// TIA Portal V20 export
// export: Created 2025-12-01T14:57:42.6383324Z, ExportSetting None, DisplayName Totally Integrated Automation Portal, DisplayVersion V20 Update 3, DisplayName TIA Portal Openness, DisplayVersion V20 Update 3, DisplayName TIA Portal Version Control Interface, DisplayVersion V20 Update 3, DisplayName STEP 7 Professional, DisplayVersion V20 Update 3, DisplayName STEP 7 Safety, DisplayVersion V20 Update 2, DisplayName WinCC Basic/Comfort/Advanced, DisplayVersion V20 Update 3, DisplayName WinCC Professional, DisplayVersion V20 Update 3, DisplayName WinCC Unified, DisplayVersion V20 Update 3
DATA_BLOCK "DB6_Recepcion"   // DB6
{ S7_Optimized_Access := 'FALSE' }
// stored: AutoNumber false
   VAR
      ByteLIbre_000 : Byte;
      FinLote_M1 : Bool;
      Especial_M1 : Bool;
      Bit_02_M1 : Bool;
      Retroceder_M1 : Bool;
      Retirar_M1 : Bool;
      Continuar_M1 : Bool;
      Entrar_M1 : Bool;
      EmiOK_M1 : Bool;
      FinLote_M2 : Bool;
      Especial_M2 : Bool;
      Bit_02_M2 : Bool;
      Retroceder_M2 : Bool;
      Retirar_M2 : Bool;
      Continuar_M2 : Bool;
      Entrar_M2 : Bool;
      EmiOK_M2 : Bool;
      FinLote_M3 : Bool;
      Especial_M3 : Bool;
      Bit_02_M3 : Bool;
      Retroceder_M3 : Bool;
      Retirar_M3 : Bool;
      Continuar_M3 : Bool;
      Entrar_M3 : Bool;
      EmiOK_M3 : Bool;
      FinLote_M4 : Bool;
      Especial_M4 : Bool;
      Bit_02_M4 : Bool;
      Retroceder_M4 : Bool;
      Retirar_M4 : Bool;
      Continuar_M4 : Bool;
      Entrar_M4 : Bool;
      EmiOK_M4 : Bool;
      FinLote_M5 : Bool;
      Especial_M5 : Bool;
      Bit_02_M5 : Bool;
      Retroceder_M5 : Bool;
      Retirar_M5 : Bool;
      Continuar_M5 : Bool;
      Entrar_M5 : Bool;
      EmiOK_M5 : Bool;
      FinLote_M6 : Bool;
      Especial_M6 : Bool;
      Bit_02_M6 : Bool;
      Retroceder_M6 : Bool;
      Retirar_M6 : Bool;
      Continuar_M6 : Bool;
      Entrar_M6 : Bool;
      EmiOK_M6 : Bool;
      FinLote_M7 : Bool;
      Especial_M7 : Bool;
      Bit_02_M7 : Bool;
      Retroceder_M7 : Bool;
      Retirar_M7 : Bool;
      Continuar_M7 : Bool;
      Entrar_M7 : Bool;
      EmiOK_M7 : Bool;
      FinLote_M8 : Bool;
      Especial_M8 : Bool;
      Bit_02_M8 : Bool;
      Retroceder_M8 : Bool;
      Retirar_M8 : Bool;
      Continuar_M8 : Bool;
      Entrar_M8 : Bool;
      EmiOK_M8 : Bool;
      FinLote_M9 : Bool;
      Especial_M9 : Bool;
      Bit_02_M9 : Bool;
      Retroceder_M9 : Bool;
      Retirar_M9 : Bool;
      Continuar_M9 : Bool;
      Entrar_M9 : Bool;
      EmiOK_M9 : Bool;
      FinLote_M10 : Bool;
      Especial_M10 : Bool;
      Bit_02_M10 : Bool;
      Retroceder_M10 : Bool;
      Retirar_M10 : Bool;
      Continuar_M10 : Bool;
      Entrar_M10 : Bool;
      EmiOK_M10 : Bool;
      FinLote_M11 : Bool;
      Especial_M11 : Bool;
      Bit_02_M11 : Bool;
      Retroceder_M11 : Bool;
      Retirar_M11 : Bool;
      Continuar_M11 : Bool;
      Entrar_M11 : Bool;
      EmiOK_M11 : Bool;
      FinLote_M12 : Bool;
      Especial_M12 : Bool;
      Bit_02_M12 : Bool;
      Retroceder_M12 : Bool;
      Retirar_M12 : Bool;
      Continuar_M12 : Bool;
      Entrar_M12 : Bool;
      EmiOK_M12 : Bool;
      FinLote_M13 : Bool;
      Especial_M13 : Bool;
      Bit_02_M13 : Bool;
      Retroceder_M13 : Bool;
      Retirar_M13 : Bool;
      Continuar_M13 : Bool;
      Entrar_M13 : Bool;
      EmiOK_M13 : Bool;
      FinLote_M14 : Bool;
      Especial_M14 : Bool;
      Bit_02_M14 : Bool;
      Retroceder_M14 : Bool;
      Retirar_M14 : Bool;
      Continuar_M14 : Bool;
      Entrar_M14 : Bool;
      EmiOK_M14 : Bool;
      FinLote_M15 : Bool;
      Especial_M15 : Bool;
      Bit_02_M15 : Bool;
      Retroceder_M15 : Bool;
      Retirar_M15 : Bool;
      Continuar_M15 : Bool;
      Entrar_M15 : Bool;
      EmiOK_M15 : Bool;
      FinLote_M16 : Bool;
      Especial_M16 : Bool;
      Bit_02_M16 : Bool;
      Retroceder_M16 : Bool;
      Retirar_M16 : Bool;
      Continuar_M16 : Bool;
      Entrar_M16 : Bool;
      EmiOK_M16 : Bool;
      FinLote_M17 : Bool;
      Especial_M17 : Bool;
      Bit_02_M17 : Bool;
      Retroceder_M17 : Bool;
      Retirar_M17 : Bool;
      Continuar_M17 : Bool;
      Entrar_M17 : Bool;
      EmiOK_M17 : Bool;
      FinLote_M18 : Bool;
      Especial_M18 : Bool;
      Bit_02_M18 : Bool;
      Retroceder_M18 : Bool;
      Retirar_M18 : Bool;
      Continuar_M18 : Bool;
      Entrar_M18 : Bool;
      EmiOK_M18 : Bool;
      FinLote_M19 : Bool;
      Especial_M19 : Bool;
      Bit_02_M19 : Bool;
      Retroceder_M19 : Bool;
      Retirar_M19 : Bool;
      Continuar_M19 : Bool;
      Entrar_M19 : Bool;
      EmiOK_M19 : Bool;
      FinLote_M20 : Bool;
      Especial_M20 : Bool;
      Bit_02_M20 : Bool;
      Retroceder_M20 : Bool;
      Retirar_M20 : Bool;
      Continuar_M20 : Bool;
      Entrar_M20 : Bool;
      EmiOK_M20 : Bool;
      FinLote_M21 : Bool;
      Especial_M21 : Bool;
      Bit_02_M21 : Bool;
      Retroceder_M21 : Bool;
      Retirar_M21 : Bool;
      Continuar_M21 : Bool;
      Entrar_M21 : Bool;
      EmiOK_M21 : Bool;
      FinLote_M22 : Bool;
      Especial_M22 : Bool;
      Bit_02_M22 : Bool;
      Retroceder_M22 : Bool;
      Retirar_M22 : Bool;
      Continuar_M22 : Bool;
      Entrar_M22 : Bool;
      EmiOK_M22 : Bool;
      FinLote_M23 : Bool;
      Especial_M23 : Bool;
      Bit_02_M23 : Bool;
      Retroceder_M23 : Bool;
      Retirar_M23 : Bool;
      Continuar_M23 : Bool;
      Entrar_M23 : Bool;
      EmiOK_M23 : Bool;
      FinLote_M24 : Bool;
      Especial_M24 : Bool;
      Bit_02_M24 : Bool;
      Retroceder_M24 : Bool;
      Retirar_M24 : Bool;
      Continuar_M24 : Bool;
      Entrar_M24 : Bool;
      EmiOK_M24 : Bool;
      FinLote_M25 : Bool;
      Especial_M25 : Bool;
      Bit_02_M25 : Bool;
      Retroceder_M25 : Bool;
      Retirar_M25 : Bool;
      Continuar_M25 : Bool;
      Entrar_M25 : Bool;
      EmiOK_M25 : Bool;
      FinLote_M26 : Bool;
      Especial_M26 : Bool;
      Bit_02_M26 : Bool;
      Retroceder_M26 : Bool;
      Retirar_M26 : Bool;
      Continuar_M26 : Bool;
      Entrar_M26 : Bool;
      EmiOK_M26 : Bool;
      FinLote_M27 : Bool;
      Especial_M27 : Bool;
      Bit_02_M27 : Bool;
      Retroceder_M27 : Bool;
      Retirar_M27 : Bool;
      Continuar_M27 : Bool;
      Entrar_M27 : Bool;
      EmiOK_M27 : Bool;
      FinLote_M28 : Bool;
      Especial_M28 : Bool;
      Bit_02_M28 : Bool;
      Retroceder_M28 : Bool;
      Retirar_M28 : Bool;
      Continuar_M28 : Bool;
      Entrar_M28 : Bool;
      EmiOK_M28 : Bool;
      FinLote_M29 : Bool;
      Especial_M29 : Bool;
      Bit_02_M29 : Bool;
      Retroceder_M29 : Bool;
      Retirar_M29 : Bool;
      Continuar_M29 : Bool;
      Entrar_M29 : Bool;
      EmiOK_M29 : Bool;
      FinLote_M30 : Bool;
      Especial_M30 : Bool;
      Bit_02_M30 : Bool;
      Retroceder_M30 : Bool;
      Retirar_M30 : Bool;
      Continuar_M30 : Bool;
      Entrar_M30 : Bool;
      EmiOK_M30 : Bool;
      FinLote_M31 : Bool;
      Especial_M31 : Bool;
      Bit_02_M31 : Bool;
      Retroceder_M31 : Bool;
      Retirar_M31 : Bool;
      Continuar_M31 : Bool;
      Entrar_M31 : Bool;
      EmiOK_M31 : Bool;
      FinLote_M32 : Bool;
      Especial_M32 : Bool;
      Bit_02_M32 : Bool;
      Retroceder_M32 : Bool;
      Retirar_M32 : Bool;
      Continuar_M32 : Bool;
      Entrar_M32 : Bool;
      EmiOK_M32 : Bool;
      FinLote_M33 : Bool;
      Especial_M33 : Bool;
      Bit_02_M33 : Bool;
      Retroceder_M33 : Bool;
      Retirar_M33 : Bool;
      Continuar_M33 : Bool;
      Entrar_M33 : Bool;
      EmiOK_M33 : Bool;
      FinLote_M34 : Bool;
      Especial_M34 : Bool;
      Bit_02_M34 : Bool;
      Retroceder_M34 : Bool;
      Retirar_M34 : Bool;
      Continuar_M34 : Bool;
      Entrar_M34 : Bool;
      EmiOK_M34 : Bool;
      FinLote_M35 : Bool;
      Especial_M35 : Bool;
      Bit_02_M35 : Bool;
      Retroceder_M35 : Bool;
      Retirar_M35 : Bool;
      Continuar_M35 : Bool;
      Entrar_M35 : Bool;
      EmiOK_M35 : Bool;
      FinLote_M36 : Bool;
      Especial_M36 : Bool;
      Bit_02_M36 : Bool;
      Retroceder_M36 : Bool;
      Retirar_M36 : Bool;
      Continuar_M36 : Bool;
      Entrar_M36 : Bool;
      EmiOK_M36 : Bool;
      FinLote_M37 : Bool;
      Especial_M37 : Bool;
      Bit_02_M37 : Bool;
      Retroceder_M37 : Bool;
      Retirar_M37 : Bool;
      Continuar_M37 : Bool;
      Entrar_M37 : Bool;
      EmiOK_M37 : Bool;
      FinLote_M38 : Bool;
      Especial_M38 : Bool;
      Bit_02_M38 : Bool;
      Retroceder_M38 : Bool;
      Retirar_M38 : Bool;
      Continuar_M38 : Bool;
      Entrar_M38 : Bool;
      EmiOK_M38 : Bool;
      FinLote_M39 : Bool;
      Especial_M39 : Bool;
      Bit_02_M39 : Bool;
      Retroceder_M39 : Bool;
      Retirar_M39 : Bool;
      Continuar_M39 : Bool;
      Entrar_M39 : Bool;
      EmiOK_M39 : Bool;
      FinLote_M40 : Bool;
      Especial_M40 : Bool;
      Bit_02_M40 : Bool;
      Retroceder_M40 : Bool;
      Retirar_M40 : Bool;
      Continuar_M40 : Bool;
      Entrar_M40 : Bool;
      EmiOK_M40 : Bool;
      FinLote_M41 : Bool;
      Especial_M41 : Bool;
      Bit_02_M41 : Bool;
      Retroceder_M41 : Bool;
      Retirar_M41 : Bool;
      Continuar_M41 : Bool;
      Entrar_M41 : Bool;
      EmiOK_M41 : Bool;
      FinLote_M42 : Bool;
      Especial_M42 : Bool;
      Bit_02_M42 : Bool;
      Retroceder_M42 : Bool;
      Retirar_M42 : Bool;
      Continuar_M42 : Bool;
      Entrar_M42 : Bool;
      EmiOK_M42 : Bool;
      FinLote_M43 : Bool;
      Especial_M43 : Bool;
      Bit_02_M43 : Bool;
      Retroceder_M43 : Bool;
      Retirar_M43 : Bool;
      Continuar_M43 : Bool;
      Entrar_M43 : Bool;
      EmiOK_M43 : Bool;
      FinLote_M44 : Bool;
      Especial_M44 : Bool;
      Bit_02_M44 : Bool;
      Retroceder_M44 : Bool;
      Retirar_M44 : Bool;
      Continuar_M44 : Bool;
      Entrar_M44 : Bool;
      EmiOK_M44 : Bool;
      FinLote_M45 : Bool;
      Especial_M45 : Bool;
      Bit_02_M45 : Bool;
      Retroceder_M45 : Bool;
      Retirar_M45 : Bool;
      Continuar_M45 : Bool;
      Entrar_M45 : Bool;
      EmiOK_M45 : Bool;
      FinLote_M46 : Bool;
      Especial_M46 : Bool;
      Bit_02_M46 : Bool;
      Retroceder_M46 : Bool;
      Retirar_M46 : Bool;
      Continuar_M46 : Bool;
      Entrar_M46 : Bool;
      EmiOK_M46 : Bool;
      FinLote_M47 : Bool;
      Especial_M47 : Bool;
      Bit_02_M47 : Bool;
      Retroceder_M47 : Bool;
      Retirar_M47 : Bool;
      Continuar_M47 : Bool;
      Entrar_M47 : Bool;
      EmiOK_M47 : Bool;
      FinLote_M48 : Bool;
      Especial_M48 : Bool;
      Bit_02_M48 : Bool;
      Retroceder_M48 : Bool;
      Retirar_M48 : Bool;
      Continuar_M48 : Bool;
      Entrar_M48 : Bool;
      EmiOK_M48 : Bool;
      FinLote_M49 : Bool;
      Especial_M49 : Bool;
      Bit_02_M49 : Bool;
      Retroceder_M49 : Bool;
      Retirar_M49 : Bool;
      Continuar_M49 : Bool;
      Entrar_M49 : Bool;
      EmiOK_M49 : Bool;
      FinLote_M50 : Bool;
      Especial_M50 : Bool;
      Bit_02_M50 : Bool;
      Retroceder_M50 : Bool;
      Retirar_M50 : Bool;
      Continuar_M50 : Bool;
      Entrar_M50 : Bool;
      EmiOK_M50 : Bool;
      FinLote_M51 : Bool;
      Especial_M51 : Bool;
      Bit_02_M51 : Bool;
      Retroceder_M51 : Bool;
      Retirar_M51 : Bool;
      Continuar_M51 : Bool;
      Entrar_M51 : Bool;
      EmiOK_M51 : Bool;
      FinLote_M52 : Bool;
      Especial_M52 : Bool;
      Bit_02_M52 : Bool;
      Retroceder_M52 : Bool;
      Retirar_M52 : Bool;
      Continuar_M52 : Bool;
      Entrar_M52 : Bool;
      EmiOK_M52 : Bool;
      FinLote_M53 : Bool;
      Especial_M53 : Bool;
      Bit_02_M53 : Bool;
      Retroceder_M53 : Bool;
      Retirar_M53 : Bool;
      Continuar_M53 : Bool;
      Entrar_M53 : Bool;
      EmiOK_M53 : Bool;
      FinLote_M54 : Bool;
      Especial_M54 : Bool;
      Bit_02_M54 : Bool;
      Retroceder_M54 : Bool;
      Retirar_M54 : Bool;
      Continuar_M54 : Bool;
      Entrar_M54 : Bool;
      EmiOK_M54 : Bool;
      FinLote_M55 : Bool;
      Especial_M55 : Bool;
      Bit_02_M55 : Bool;
      Retroceder_M55 : Bool;
      Retirar_M55 : Bool;
      Continuar_M55 : Bool;
      Entrar_M55 : Bool;
      EmiOK_M55 : Bool;
      FinLote_M56 : Bool;
      Especial_M56 : Bool;
      Bit_02_M56 : Bool;
      Retroceder_M56 : Bool;
      Retirar_M56 : Bool;
      Continuar_M56 : Bool;
      Entrar_M56 : Bool;
      EmiOK_M56 : Bool;
      FinLote_M57 : Bool;
      Especial_M57 : Bool;
      Bit_02_M57 : Bool;
      Retroceder_M57 : Bool;
      Retirar_M57 : Bool;
      Continuar_M57 : Bool;
      Entrar_M57 : Bool;
      EmiOK_M57 : Bool;
      FinLote_M58 : Bool;
      Especial_M58 : Bool;
      Bit_02_M58 : Bool;
      Retroceder_M58 : Bool;
      Retirar_M58 : Bool;
      Continuar_M58 : Bool;
      Entrar_M58 : Bool;
      EmiOK_M58 : Bool;
      FinLote_M59 : Bool;
      Especial_M59 : Bool;
      Bit_02_M59 : Bool;
      Retroceder_M59 : Bool;
      Retirar_M59 : Bool;
      Continuar_M59 : Bool;
      Entrar_M59 : Bool;
      EmiOK_M59 : Bool;
      FinLote_M60 : Bool;
      Especial_M60 : Bool;
      Bit_02_M60 : Bool;
      Retroceder_M60 : Bool;
      Retirar_M60 : Bool;
      Continuar_M60 : Bool;
      Entrar_M60 : Bool;
      EmiOK_M60 : Bool;
      FinLote_M61 : Bool;
      Especial_M61 : Bool;
      Bit_02_M61 : Bool;
      Retroceder_M61 : Bool;
      Retirar_M61 : Bool;
      Continuar_M61 : Bool;
      Entrar_M61 : Bool;
      EmiOK_M61 : Bool;
      FinLote_M62 : Bool;
      Especial_M62 : Bool;
      Bit_02_M62 : Bool;
      Retroceder_M62 : Bool;
      Retirar_M62 : Bool;
      Continuar_M62 : Bool;
      Entrar_M62 : Bool;
      EmiOK_M62 : Bool;
      FinLote_M63 : Bool;
      Especial_M63 : Bool;
      Bit_02_M63 : Bool;
      Retroceder_M63 : Bool;
      Retirar_M63 : Bool;
      Continuar_M63 : Bool;
      Entrar_M63 : Bool;
      EmiOK_M63 : Bool;
      FinLote_M64 : Bool;
      Especial_M64 : Bool;
      Bit_02_M64 : Bool;
      Retroceder_M64 : Bool;
      Retirar_M64 : Bool;
      Continuar_M64 : Bool;
      Entrar_M64 : Bool;
      EmiOK_M64 : Bool;
      FinLote_M65 : Bool;
      Especial_M65 : Bool;
      Bit_02_M65 : Bool;
      Retroceder_M65 : Bool;
      Retirar_M65 : Bool;
      Continuar_M65 : Bool;
      Entrar_M65 : Bool;
      EmiOK_M65 : Bool;
      FinLote_M66 : Bool;
      Especial_M66 : Bool;
      Bit_02_M66 : Bool;
      Retroceder_M66 : Bool;
      Retirar_M66 : Bool;
      Continuar_M66 : Bool;
      Entrar_M66 : Bool;
      EmiOK_M66 : Bool;
      FinLote_M67 : Bool;
      Especial_M67 : Bool;
      Bit_02_M67 : Bool;
      Retroceder_M67 : Bool;
      Retirar_M67 : Bool;
      Continuar_M67 : Bool;
      Entrar_M67 : Bool;
      EmiOK_M67 : Bool;
      FinLote_M68 : Bool;
      Especial_M68 : Bool;
      Bit_02_M68 : Bool;
      Retroceder_M68 : Bool;
      Retirar_M68 : Bool;
      Continuar_M68 : Bool;
      Entrar_M68 : Bool;
      EmiOK_M68 : Bool;
      FinLote_M69 : Bool;
      Especial_M69 : Bool;
      Bit_02_M69 : Bool;
      Retroceder_M69 : Bool;
      Retirar_M69 : Bool;
      Continuar_M69 : Bool;
      Entrar_M69 : Bool;
      EmiOK_M69 : Bool;
      FinLote_M70 : Bool;
      Especial_M70 : Bool;
      Bit_02_M70 : Bool;
      Retroceder_M70 : Bool;
      Retirar_M70 : Bool;
      Continuar_M70 : Bool;
      Entrar_M70 : Bool;
      EmiOK_M70 : Bool;
      FinLote_M71 : Bool;
      Especial_M71 : Bool;
      Bit_02_M71 : Bool;
      Retroceder_M71 : Bool;
      Retirar_M71 : Bool;
      Continuar_M71 : Bool;
      Entrar_M71 : Bool;
      EmiOK_M71 : Bool;
      FinLote_M72 : Bool;
      Especial_M72 : Bool;
      Bit_02_M72 : Bool;
      Retroceder_M72 : Bool;
      Retirar_M72 : Bool;
      Continuar_M72 : Bool;
      Entrar_M72 : Bool;
      EmiOK_M72 : Bool;
      FinLote_M73 : Bool;
      Especial_M73 : Bool;
      Bit_02_M73 : Bool;
      Retroceder_M73 : Bool;
      Retirar_M73 : Bool;
      Continuar_M73 : Bool;
      Entrar_M73 : Bool;
      EmiOK_M73 : Bool;
      FinLote_M74 : Bool;
      Especial_M74 : Bool;
      Bit_02_M74 : Bool;
      Retroceder_M74 : Bool;
      Retirar_M74 : Bool;
      Continuar_M74 : Bool;
      Entrar_M74 : Bool;
      EmiOK_M74 : Bool;
      FinLote_M75 : Bool;
      Especial_M75 : Bool;
      Bit_02_M75 : Bool;
      Retroceder_M75 : Bool;
      Retirar_M75 : Bool;
      Continuar_M75 : Bool;
      Entrar_M75 : Bool;
      EmiOK_M75 : Bool;
      FinLote_M76 : Bool;
      Especial_M76 : Bool;
      Bit_02_M76 : Bool;
      Retroceder_M76 : Bool;
      Retirar_M76 : Bool;
      Continuar_M76 : Bool;
      Entrar_M76 : Bool;
      EmiOK_M76 : Bool;
      FinLote_M77 : Bool;
      Especial_M77 : Bool;
      Bit_02_M77 : Bool;
      Retroceder_M77 : Bool;
      Retirar_M77 : Bool;
      Continuar_M77 : Bool;
      Entrar_M77 : Bool;
      EmiOK_M77 : Bool;
      FinLote_M78 : Bool;
      Especial_M78 : Bool;
      Bit_02_M78 : Bool;
      Retroceder_M78 : Bool;
      Retirar_M78 : Bool;
      Continuar_M78 : Bool;
      Entrar_M78 : Bool;
      EmiOK_M78 : Bool;
      FinLote_M79 : Bool;
      Especial_M79 : Bool;
      Bit_02_M79 : Bool;
      Retroceder_M79 : Bool;
      Retirar_M79 : Bool;
      Continuar_M79 : Bool;
      Entrar_M79 : Bool;
      EmiOK_M79 : Bool;
      FinLote_M80 : Bool;
      Especial_M80 : Bool;
      Bit_02_M80 : Bool;
      Retroceder_M80 : Bool;
      Retirar_M80 : Bool;
      Continuar_M80 : Bool;
      Entrar_M80 : Bool;
      EmiOK_M80 : Bool;
      FinLote_M81 : Bool;
      Especial_M81 : Bool;
      Bit_02_M81 : Bool;
      Retroceder_M81 : Bool;
      Retirar_M81 : Bool;
      Continuar_M81 : Bool;
      Entrar_M81 : Bool;
      EmiOK_M81 : Bool;
      FinLote_M82 : Bool;
      Especial_M82 : Bool;
      Bit_02_M82 : Bool;
      Retroceder_M82 : Bool;
      Retirar_M82 : Bool;
      Continuar_M82 : Bool;
      Entrar_M82 : Bool;
      EmiOK_M82 : Bool;
      FinLote_M83 : Bool;
      Especial_M83 : Bool;
      Bit_02_M83 : Bool;
      Retroceder_M83 : Bool;
      Retirar_M83 : Bool;
      Continuar_M83 : Bool;
      Entrar_M83 : Bool;
      EmiOK_M83 : Bool;
      FinLote_M84 : Bool;
      Especial_M84 : Bool;
      Bit_02_M84 : Bool;
      Retroceder_M84 : Bool;
      Retirar_M84 : Bool;
      Continuar_M84 : Bool;
      Entrar_M84 : Bool;
      EmiOK_M84 : Bool;
      FinLote_M85 : Bool;
      Especial_M85 : Bool;
      Bit_02_M85 : Bool;
      Retroceder_M85 : Bool;
      Retirar_M85 : Bool;
      Continuar_M85 : Bool;
      Entrar_M85 : Bool;
      EmiOK_M85 : Bool;
      FinLote_M86 : Bool;
      Especial_M86 : Bool;
      Bit_02_M86 : Bool;
      Retroceder_M86 : Bool;
      Retirar_M86 : Bool;
      Continuar_M86 : Bool;
      Entrar_M86 : Bool;
      EmiOK_M86 : Bool;
      FinLote_M87 : Bool;
      Especial_M87 : Bool;
      Bit_02_M87 : Bool;
      Retroceder_M87 : Bool;
      Retirar_M87 : Bool;
      Continuar_M87 : Bool;
      Entrar_M87 : Bool;
      EmiOK_M87 : Bool;
      FinLote_M88 : Bool;
      Especial_M88 : Bool;
      Bit_02_M88 : Bool;
      Retroceder_M88 : Bool;
      Retirar_M88 : Bool;
      Continuar_M88 : Bool;
      Entrar_M88 : Bool;
      EmiOK_M88 : Bool;
      FinLote_M89 : Bool;
      Especial_M89 : Bool;
      Bit_02_M89 : Bool;
      Retroceder_M89 : Bool;
      Retirar_M89 : Bool;
      Continuar_M89 : Bool;
      Entrar_M89 : Bool;
      EmiOK_M89 : Bool;
      FinLote_M90 : Bool;
      Especial_M90 : Bool;
      Bit_02_M90 : Bool;
      Retroceder_M90 : Bool;
      Retirar_M90 : Bool;
      Continuar_M90 : Bool;
      Entrar_M90 : Bool;
      EmiOK_M90 : Bool;
      FinLote_M91 : Bool;
      Especial_M91 : Bool;
      Bit_02_M91 : Bool;
      Retroceder_M91 : Bool;
      Retirar_M91 : Bool;
      Continuar_M91 : Bool;
      Entrar_M91 : Bool;
      EmiOK_M91 : Bool;
      FinLote_M92 : Bool;
      Especial_M92 : Bool;
      Bit_02_M92 : Bool;
      Retroceder_M92 : Bool;
      Retirar_M92 : Bool;
      Continuar_M92 : Bool;
      Entrar_M92 : Bool;
      EmiOK_M92 : Bool;
      FinLote_M93 : Bool;
      Especial_M93 : Bool;
      Bit_02_M93 : Bool;
      Retroceder_M93 : Bool;
      Retirar_M93 : Bool;
      Continuar_M93 : Bool;
      Entrar_M93 : Bool;
      EmiOK_M93 : Bool;
      FinLote_M94 : Bool;
      Especial_M94 : Bool;
      Bit_02_M94 : Bool;
      Retroceder_M94 : Bool;
      Retirar_M94 : Bool;
      Continuar_M94 : Bool;
      Entrar_M94 : Bool;
      EmiOK_M94 : Bool;
      FinLote_M95 : Bool;
      Especial_M95 : Bool;
      Bit_02_M95 : Bool;
      Retroceder_M95 : Bool;
      Retirar_M95 : Bool;
      Continuar_M95 : Bool;
      Entrar_M95 : Bool;
      EmiOK_M95 : Bool;
      FinLote_M96 : Bool;
      Especial_M96 : Bool;
      Bit_02_M96 : Bool;
      Retroceder_M96 : Bool;
      Retirar_M96 : Bool;
      Continuar_M96 : Bool;
      Entrar_M96 : Bool;
      EmiOK_M96 : Bool;
      FinLote_M97 : Bool;
      Especial_M97 : Bool;
      Bit_02_M97 : Bool;
      Retroceder_M97 : Bool;
      Retirar_M97 : Bool;
      Continuar_M97 : Bool;
      Entrar_M97 : Bool;
      EmiOK_M97 : Bool;
      FinLote_M98 : Bool;
      Especial_M98 : Bool;
      Bit_02_M98 : Bool;
      Retroceder_M98 : Bool;
      Retirar_M98 : Bool;
      Continuar_M98 : Bool;
      Entrar_M98 : Bool;
      EmiOK_M98 : Bool;
      FinLote_M99 : Bool;
      Especial_M99 : Bool;
      Bit_02_M99 : Bool;
      Retroceder_M99 : Bool;
      Retirar_M99 : Bool;
      Continuar_M99 : Bool;
      Entrar_M99 : Bool;
      EmiOK_M99 : Bool;
      FinLote_M100 : Bool;
      Especial_M100 : Bool;
      Bit_02_M100 : Bool;
      Retroceder_M100 : Bool;
      Retirar_M100 : Bool;
      Continuar_M100 : Bool;
      Entrar_M100 : Bool;
      EmiOK_M100 : Bool;
      FinLote_M101 : Bool;
      Especial_M101 : Bool;
      Bit_02_M101 : Bool;
      Retroceder_M101 : Bool;
      Retirar_M101 : Bool;
      Continuar_M101 : Bool;
      Entrar_M101 : Bool;
      EmiOK_M101 : Bool;
      FinLote_M102 : Bool;
      Especial_M102 : Bool;
      Bit_02_M102 : Bool;
      Retroceder_M102 : Bool;
      Retirar_M102 : Bool;
      Continuar_M102 : Bool;
      Entrar_M102 : Bool;
      EmiOK_M102 : Bool;
      FinLote_M103 : Bool;
      Especial_M103 : Bool;
      Bit_02_M103 : Bool;
      Retroceder_M103 : Bool;
      Retirar_M103 : Bool;
      Continuar_M103 : Bool;
      Entrar_M103 : Bool;
      EmiOK_M103 : Bool;
      FinLote_M104 : Bool;
      Especial_M104 : Bool;
      Bit_02_M104 : Bool;
      Retroceder_M104 : Bool;
      Retirar_M104 : Bool;
      Continuar_M104 : Bool;
      Entrar_M104 : Bool;
      EmiOK_M104 : Bool;
      FinLote_M105 : Bool;
      Especial_M105 : Bool;
      Bit_02_M105 : Bool;
      Retroceder_M105 : Bool;
      Retirar_M105 : Bool;
      Continuar_M105 : Bool;
      Entrar_M105 : Bool;
      EmiOK_M105 : Bool;
      FinLote_M106 : Bool;
      Especial_M106 : Bool;
      Bit_02_M106 : Bool;
      Retroceder_M106 : Bool;
      Retirar_M106 : Bool;
      Continuar_M106 : Bool;
      Entrar_M106 : Bool;
      EmiOK_M106 : Bool;
      FinLote_M107 : Bool;
      Especial_M107 : Bool;
      Bit_02_M107 : Bool;
      Retroceder_M107 : Bool;
      Retirar_M107 : Bool;
      Continuar_M107 : Bool;
      Entrar_M107 : Bool;
      EmiOK_M107 : Bool;
      FinLote_M108 : Bool;
      Especial_M108 : Bool;
      Bit_02_M108 : Bool;
      Retroceder_M108 : Bool;
      Retirar_M108 : Bool;
      Continuar_M108 : Bool;
      Entrar_M108 : Bool;
      EmiOK_M108 : Bool;
      FinLote_M109 : Bool;
      Especial_M109 : Bool;
      Bit_02_M109 : Bool;
      Retroceder_M109 : Bool;
      Retirar_M109 : Bool;
      Continuar_M109 : Bool;
      Entrar_M109 : Bool;
      EmiOK_M109 : Bool;
      FinLote_M110 : Bool;
      Especial_M110 : Bool;
      Bit_02_M110 : Bool;
      Retroceder_M110 : Bool;
      Retirar_M110 : Bool;
      Continuar_M110 : Bool;
      Entrar_M110 : Bool;
      EmiOK_M110 : Bool;
      FinLote_M111 : Bool;
      Especial_M111 : Bool;
      Bit_02_M111 : Bool;
      Retroceder_M111 : Bool;
      Retirar_M111 : Bool;
      Continuar_M111 : Bool;
      Entrar_M111 : Bool;
      EmiOK_M111 : Bool;
      FinLote_M112 : Bool;
      Especial_M112 : Bool;
      Bit_02_M112 : Bool;
      Retroceder_M112 : Bool;
      Retirar_M112 : Bool;
      Continuar_M112 : Bool;
      Entrar_M112 : Bool;
      EmiOK_M112 : Bool;
      FinLote_M113 : Bool;
      Especial_M113 : Bool;
      Bit_02_M113 : Bool;
      Retroceder_M113 : Bool;
      Retirar_M113 : Bool;
      Continuar_M113 : Bool;
      Entrar_M113 : Bool;
      EmiOK_M113 : Bool;
      FinLote_M114 : Bool;
      Especial_M114 : Bool;
      Bit_02_M114 : Bool;
      Retroceder_M114 : Bool;
      Retirar_M114 : Bool;
      Continuar_M114 : Bool;
      Entrar_M114 : Bool;
      EmiOK_M114 : Bool;
      FinLote_M115 : Bool;
      Especial_M115 : Bool;
      Bit_02_M115 : Bool;
      Retroceder_M115 : Bool;
      Retirar_M115 : Bool;
      Continuar_M115 : Bool;
      Entrar_M115 : Bool;
      EmiOK_M115 : Bool;
      FinLote_M116 : Bool;
      Especial_M116 : Bool;
      Bit_02_M116 : Bool;
      Retroceder_M116 : Bool;
      Retirar_M116 : Bool;
      Continuar_M116 : Bool;
      Entrar_M116 : Bool;
      EmiOK_M116 : Bool;
      FinLote_M117 : Bool;
      Especial_M117 : Bool;
      Bit_02_M117 : Bool;
      Retroceder_M117 : Bool;
      Retirar_M117 : Bool;
      Continuar_M117 : Bool;
      Entrar_M117 : Bool;
      EmiOK_M117 : Bool;
      FinLote_M118 : Bool;
      Especial_M118 : Bool;
      Bit_02_M118 : Bool;
      Retroceder_M118 : Bool;
      Retirar_M118 : Bool;
      Continuar_M118 : Bool;
      Entrar_M118 : Bool;
      EmiOK_M118 : Bool;
      FinLote_M119 : Bool;
      Especial_M119 : Bool;
      Bit_02_M119 : Bool;
      Retroceder_M119 : Bool;
      Retirar_M119 : Bool;
      Continuar_M119 : Bool;
      Entrar_M119 : Bool;
      EmiOK_M119 : Bool;
      FinLote_M120 : Bool;
      Especial_M120 : Bool;
      Bit_02_M120 : Bool;
      Retroceder_M120 : Bool;
      Retirar_M120 : Bool;
      Continuar_M120 : Bool;
      Entrar_M120 : Bool;
      EmiOK_M120 : Bool;
      FinLote_M121 : Bool;
      Especial_M121 : Bool;
      Bit_02_M121 : Bool;
      Retroceder_M121 : Bool;
      Retirar_M121 : Bool;
      Continuar_M121 : Bool;
      Entrar_M121 : Bool;
      EmiOK_M121 : Bool;
      FinLote_M122 : Bool;
      Especial_M122 : Bool;
      Bit_02_M122 : Bool;
      Retroceder_M122 : Bool;
      Retirar_M122 : Bool;
      Continuar_M122 : Bool;
      Entrar_M122 : Bool;
      EmiOK_M122 : Bool;
      FinLote_M123 : Bool;
      Especial_M123 : Bool;
      Bit_02_M123 : Bool;
      Retroceder_M123 : Bool;
      Retirar_M123 : Bool;
      Continuar_M123 : Bool;
      Entrar_M123 : Bool;
      EmiOK_M123 : Bool;
      FinLote_M124 : Bool;
      Especial_M124 : Bool;
      Bit_02_M124 : Bool;
      Retroceder_M124 : Bool;
      Retirar_M124 : Bool;
      Continuar_M124 : Bool;
      Entrar_M124 : Bool;
      EmiOK_M124 : Bool;
      FinLote_M125 : Bool;
      Especial_M125 : Bool;
      Bit_02_M125 : Bool;
      Retroceder_M125 : Bool;
      Retirar_M125 : Bool;
      Continuar_M125 : Bool;
      Entrar_M125 : Bool;
      EmiOK_M125 : Bool;
      FinLote_M126 : Bool;
      Especial_M126 : Bool;
      Bit_02_M126 : Bool;
      Retroceder_M126 : Bool;
      Retirar_M126 : Bool;
      Continuar_M126 : Bool;
      Entrar_M126 : Bool;
      EmiOK_M126 : Bool;
      FinLote_M127 : Bool;
      Especial_M127 : Bool;
      Bit_02_M127 : Bool;
      Retroceder_M127 : Bool;
      Retirar_M127 : Bool;
      Continuar_M127 : Bool;
      Entrar_M127 : Bool;
      EmiOK_M127 : Bool;
      FinLote_M128 : Bool;
      Especial_M128 : Bool;
      Bit_02_M128 : Bool;
      Retroceder_M128 : Bool;
      Retirar_M128 : Bool;
      Continuar_M128 : Bool;
      Entrar_M128 : Bool;
      EmiOK_M128 : Bool;
      FinLote_M129 : Bool;
      Especial_M129 : Bool;
      Bit_02_M129 : Bool;
      Retroceder_M129 : Bool;
      Retirar_M129 : Bool;
      Continuar_M129 : Bool;
      Entrar_M129 : Bool;
      EmiOK_M129 : Bool;
      FinLote_M130 : Bool;
      Especial_M130 : Bool;
      Bit_02_M130 : Bool;
      Retroceder_M130 : Bool;
      Retirar_M130 : Bool;
      Continuar_M130 : Bool;
      Entrar_M130 : Bool;
      EmiOK_M130 : Bool;
      FinLote_M131 : Bool;
      Especial_M131 : Bool;
      Bit_02_M131 : Bool;
      Retroceder_M131 : Bool;
      Retirar_M131 : Bool;
      Continuar_M131 : Bool;
      Entrar_M131 : Bool;
      EmiOK_M131 : Bool;
      FinLote_M132 : Bool;
      Especial_M132 : Bool;
      Bit_02_M132 : Bool;
      Retroceder_M132 : Bool;
      Retirar_M132 : Bool;
      Continuar_M132 : Bool;
      Entrar_M132 : Bool;
      EmiOK_M132 : Bool;
      FinLote_M133 : Bool;
      Especial_M133 : Bool;
      Bit_02_M133 : Bool;
      Retroceder_M133 : Bool;
      Retirar_M133 : Bool;
      Continuar_M133 : Bool;
      Entrar_M133 : Bool;
      EmiOK_M133 : Bool;
      FinLote_M134 : Bool;
      Especial_M134 : Bool;
      Bit_02_M134 : Bool;
      Retroceder_M134 : Bool;
      Retirar_M134 : Bool;
      Continuar_M134 : Bool;
      Entrar_M134 : Bool;
      EmiOK_M134 : Bool;
      FinLote_M135 : Bool;
      Especial_M135 : Bool;
      Bit_02_M135 : Bool;
      Retroceder_M135 : Bool;
      Retirar_M135 : Bool;
      Continuar_M135 : Bool;
      Entrar_M135 : Bool;
      EmiOK_M135 : Bool;
      FinLote_M136 : Bool;
      Especial_M136 : Bool;
      Bit_02_M136 : Bool;
      Retroceder_M136 : Bool;
      Retirar_M136 : Bool;
      Continuar_M136 : Bool;
      Entrar_M136 : Bool;
      EmiOK_M136 : Bool;
      FinLote_M137 : Bool;
      Especial_M137 : Bool;
      Bit_02_M137 : Bool;
      Retroceder_M137 : Bool;
      Retirar_M137 : Bool;
      Continuar_M137 : Bool;
      Entrar_M137 : Bool;
      EmiOK_M137 : Bool;
      FinLote_M138 : Bool;
      Especial_M138 : Bool;
      Bit_02_M138 : Bool;
      Retroceder_M138 : Bool;
      Retirar_M138 : Bool;
      Continuar_M138 : Bool;
      Entrar_M138 : Bool;
      EmiOK_M138 : Bool;
      FinLote_M139 : Bool;
      Especial_M139 : Bool;
      Bit_02_M139 : Bool;
      Retroceder_M139 : Bool;
      Retirar_M139 : Bool;
      Continuar_M139 : Bool;
      Entrar_M139 : Bool;
      EmiOK_M139 : Bool;
      FinLote_M140 : Bool;
      Especial_M140 : Bool;
      Bit_02_M140 : Bool;
      Retroceder_M140 : Bool;
      Retirar_M140 : Bool;
      Continuar_M140 : Bool;
      Entrar_M140 : Bool;
      EmiOK_M140 : Bool;
      FinLote_M141 : Bool;
      Especial_M141 : Bool;
      Bit_02_M141 : Bool;
      Retroceder_M141 : Bool;
      Retirar_M141 : Bool;
      Continuar_M141 : Bool;
      Entrar_M141 : Bool;
      EmiOK_M141 : Bool;
      FinLote_M142 : Bool;
      Especial_M142 : Bool;
      Bit_02_M142 : Bool;
      Retroceder_M142 : Bool;
      Retirar_M142 : Bool;
      Continuar_M142 : Bool;
      Entrar_M142 : Bool;
      EmiOK_M142 : Bool;
      FinLote_M143 : Bool;
      Especial_M143 : Bool;
      Bit_02_M143 : Bool;
      Retroceder_M143 : Bool;
      Retirar_M143 : Bool;
      Continuar_M143 : Bool;
      Entrar_M143 : Bool;
      EmiOK_M143 : Bool;
      FinLote_M144 : Bool;
      Especial_M144 : Bool;
      Bit_02_M144 : Bool;
      Retroceder_M144 : Bool;
      Retirar_M144 : Bool;
      Continuar_M144 : Bool;
      Entrar_M144 : Bool;
      EmiOK_M144 : Bool;
      FinLote_M145 : Bool;
      Especial_M145 : Bool;
      Bit_02_M145 : Bool;
      Retroceder_M145 : Bool;
      Retirar_M145 : Bool;
      Continuar_M145 : Bool;
      Entrar_M145 : Bool;
      EmiOK_M145 : Bool;
      FinLote_M146 : Bool;
      Especial_M146 : Bool;
      Bit_02_M146 : Bool;
      Retroceder_M146 : Bool;
      Retirar_M146 : Bool;
      Continuar_M146 : Bool;
      Entrar_M146 : Bool;
      EmiOK_M146 : Bool;
      FinLote_M147 : Bool;
      Especial_M147 : Bool;
      Bit_02_M147 : Bool;
      Retroceder_M147 : Bool;
      Retirar_M147 : Bool;
      Continuar_M147 : Bool;
      Entrar_M147 : Bool;
      EmiOK_M147 : Bool;
      FinLote_M148 : Bool;
      Especial_M148 : Bool;
      Bit_02_M148 : Bool;
      Retroceder_M148 : Bool;
      Retirar_M148 : Bool;
      Continuar_M148 : Bool;
      Entrar_M148 : Bool;
      EmiOK_M148 : Bool;
      FinLote_M149 : Bool;
      Especial_M149 : Bool;
      Bit_02_M149 : Bool;
      Retroceder_M149 : Bool;
      Retirar_M149 : Bool;
      Continuar_M149 : Bool;
      Entrar_M149 : Bool;
      EmiOK_M149 : Bool;
      FinLote_M150 : Bool;
      Especial_M150 : Bool;
      Bit_02_M150 : Bool;
      Retroceder_M150 : Bool;
      Retirar_M150 : Bool;
      Continuar_M150 : Bool;
      Entrar_M150 : Bool;
      EmiOK_M150 : Bool;
      FinLote_M151 : Bool;
      Especial_M151 : Bool;
      Bit_02_M151 : Bool;
      Retroceder_M151 : Bool;
      Retirar_M151 : Bool;
      Continuar_M151 : Bool;
      Entrar_M151 : Bool;
      EmiOK_M151 : Bool;
      FinLote_M152 : Bool;
      Especial_M152 : Bool;
      Bit_02_M152 : Bool;
      Retroceder_M152 : Bool;
      Retirar_M152 : Bool;
      Continuar_M152 : Bool;
      Entrar_M152 : Bool;
      EmiOK_M152 : Bool;
      FinLote_M153 : Bool;
      Especial_M153 : Bool;
      Bit_02_M153 : Bool;
      Retroceder_M153 : Bool;
      Retirar_M153 : Bool;
      Continuar_M153 : Bool;
      Entrar_M153 : Bool;
      EmiOK_M153 : Bool;
      FinLote_M154 : Bool;
      Especial_M154 : Bool;
      Bit_02_M154 : Bool;
      Retroceder_M154 : Bool;
      Retirar_M154 : Bool;
      Continuar_M154 : Bool;
      Entrar_M154 : Bool;
      EmiOK_M154 : Bool;
      FinLote_M155 : Bool;
      Especial_M155 : Bool;
      Bit_02_M155 : Bool;
      Retroceder_M155 : Bool;
      Retirar_M155 : Bool;
      Continuar_M155 : Bool;
      Entrar_M155 : Bool;
      EmiOK_M155 : Bool;
      FinLote_M156 : Bool;
      Especial_M156 : Bool;
      Bit_02_M156 : Bool;
      Retroceder_M156 : Bool;
      Retirar_M156 : Bool;
      Continuar_M156 : Bool;
      Entrar_M156 : Bool;
      EmiOK_M156 : Bool;
      FinLote_M157 : Bool;
      Especial_M157 : Bool;
      Bit_02_M157 : Bool;
      Retroceder_M157 : Bool;
      Retirar_M157 : Bool;
      Continuar_M157 : Bool;
      Entrar_M157 : Bool;
      EmiOK_M157 : Bool;
      FinLote_M158 : Bool;
      Especial_M158 : Bool;
      Bit_02_M158 : Bool;
      Retroceder_M158 : Bool;
      Retirar_M158 : Bool;
      Continuar_M158 : Bool;
      Entrar_M158 : Bool;
      EmiOK_M158 : Bool;
      FinLote_M159 : Bool;
      Especial_M159 : Bool;
      Bit_02_M159 : Bool;
      Retroceder_M159 : Bool;
      Retirar_M159 : Bool;
      Continuar_M159 : Bool;
      Entrar_M159 : Bool;
      EmiOK_M159 : Bool;
      FinLote_M160 : Bool;
      Especial_M160 : Bool;
      Bit_02_M160 : Bool;
      Retroceder_M160 : Bool;
      Retirar_M160 : Bool;
      Continuar_M160 : Bool;
      Entrar_M160 : Bool;
      EmiOK_M160 : Bool;
      FinLote_M161 : Bool;
      Especial_M161 : Bool;
      Bit_02_M161 : Bool;
      Retroceder_M161 : Bool;
      Retirar_M161 : Bool;
      Continuar_M161 : Bool;
      Entrar_M161 : Bool;
      EmiOK_M161 : Bool;
      FinLote_M162 : Bool;
      Especial_M162 : Bool;
      Bit_02_M162 : Bool;
      Retroceder_M162 : Bool;
      Retirar_M162 : Bool;
      Continuar_M162 : Bool;
      Entrar_M162 : Bool;
      EmiOK_M162 : Bool;
      FinLote_M163 : Bool;
      Especial_M163 : Bool;
      Bit_02_M163 : Bool;
      Retroceder_M163 : Bool;
      Retirar_M163 : Bool;
      Continuar_M163 : Bool;
      Entrar_M163 : Bool;
      EmiOK_M163 : Bool;
      FinLote_M164 : Bool;
      Especial_M164 : Bool;
      Bit_02_M164 : Bool;
      Retroceder_M164 : Bool;
      Retirar_M164 : Bool;
      Continuar_M164 : Bool;
      Entrar_M164 : Bool;
      EmiOK_M164 : Bool;
      FinLote_M165 : Bool;
      Especial_M165 : Bool;
      Bit_02_M165 : Bool;
      Retroceder_M165 : Bool;
      Retirar_M165 : Bool;
      Continuar_M165 : Bool;
      Entrar_M165 : Bool;
      EmiOK_M165 : Bool;
      FinLote_M166 : Bool;
      Especial_M166 : Bool;
      Bit_02_M166 : Bool;
      Retroceder_M166 : Bool;
      Retirar_M166 : Bool;
      Continuar_M166 : Bool;
      Entrar_M166 : Bool;
      EmiOK_M166 : Bool;
      FinLote_M167 : Bool;
      Especial_M167 : Bool;
      Bit_02_M167 : Bool;
      Retroceder_M167 : Bool;
      Retirar_M167 : Bool;
      Continuar_M167 : Bool;
      Entrar_M167 : Bool;
      EmiOK_M167 : Bool;
      FinLote_M168 : Bool;
      Especial_M168 : Bool;
      Bit_02_M168 : Bool;
      Retroceder_M168 : Bool;
      Retirar_M168 : Bool;
      Continuar_M168 : Bool;
      Entrar_M168 : Bool;
      EmiOK_M168 : Bool;
      FinLote_M169 : Bool;
      Especial_M169 : Bool;
      Bit_02_M169 : Bool;
      Retroceder_M169 : Bool;
      Retirar_M169 : Bool;
      Continuar_M169 : Bool;
      Entrar_M169 : Bool;
      EmiOK_M169 : Bool;
      FinLote_M170 : Bool;
      Especial_M170 : Bool;
      Bit_02_M170 : Bool;
      Retroceder_M170 : Bool;
      Retirar_M170 : Bool;
      Continuar_M170 : Bool;
      Entrar_M170 : Bool;
      EmiOK_M170 : Bool;
      FinLote_M171 : Bool;
      Especial_M171 : Bool;
      Bit_02_M171 : Bool;
      Retroceder_M171 : Bool;
      Retirar_M171 : Bool;
      Continuar_M171 : Bool;
      Entrar_M171 : Bool;
      EmiOK_M171 : Bool;
      FinLote_M172 : Bool;
      Especial_M172 : Bool;
      Bit_02_M172 : Bool;
      Retroceder_M172 : Bool;
      Retirar_M172 : Bool;
      Continuar_M172 : Bool;
      Entrar_M172 : Bool;
      EmiOK_M172 : Bool;
      FinLote_M173 : Bool;
      Especial_M173 : Bool;
      Bit_02_M173 : Bool;
      Retroceder_M173 : Bool;
      Retirar_M173 : Bool;
      Continuar_M173 : Bool;
      Entrar_M173 : Bool;
      EmiOK_M173 : Bool;
      FinLote_M174 : Bool;
      Especial_M174 : Bool;
      Bit_02_M174 : Bool;
      Retroceder_M174 : Bool;
      Retirar_M174 : Bool;
      Continuar_M174 : Bool;
      Entrar_M174 : Bool;
      EmiOK_M174 : Bool;
      FinLote_M175 : Bool;
      Especial_M175 : Bool;
      Bit_02_M175 : Bool;
      Retroceder_M175 : Bool;
      Retirar_M175 : Bool;
      Continuar_M175 : Bool;
      Entrar_M175 : Bool;
      EmiOK_M175 : Bool;
      FinLote_M176 : Bool;
      Especial_M176 : Bool;
      Bit_02_M176 : Bool;
      Retroceder_M176 : Bool;
      Retirar_M176 : Bool;
      Continuar_M176 : Bool;
      Entrar_M176 : Bool;
      EmiOK_M176 : Bool;
      FinLote_M177 : Bool;
      Especial_M177 : Bool;
      Bit_02_M177 : Bool;
      Retroceder_M177 : Bool;
      Retirar_M177 : Bool;
      Continuar_M177 : Bool;
      Entrar_M177 : Bool;
      EmiOK_M177 : Bool;
      FinLote_M178 : Bool;
      Especial_M178 : Bool;
      Bit_02_M178 : Bool;
      Retroceder_M178 : Bool;
      Retirar_M178 : Bool;
      Continuar_M178 : Bool;
      Entrar_M178 : Bool;
      EmiOK_M178 : Bool;
      FinLote_M179 : Bool;
      Especial_M179 : Bool;
      Bit_02_M179 : Bool;
      Retroceder_M179 : Bool;
      Retirar_M179 : Bool;
      Continuar_M179 : Bool;
      Entrar_M179 : Bool;
      EmiOK_M179 : Bool;
      FinLote_M180 : Bool;
      Especial_M180 : Bool;
      Bit_02_M180 : Bool;
      Retroceder_M180 : Bool;
      Retirar_M180 : Bool;
      Continuar_M180 : Bool;
      Entrar_M180 : Bool;
      EmiOK_M180 : Bool;
      FinLote_M181 : Bool;
      Especial_M181 : Bool;
      Bit_02_M181 : Bool;
      Retroceder_M181 : Bool;
      Retirar_M181 : Bool;
      Continuar_M181 : Bool;
      Entrar_M181 : Bool;
      EmiOK_M181 : Bool;
      FinLote_M182 : Bool;
      Especial_M182 : Bool;
      Bit_02_M182 : Bool;
      Retroceder_M182 : Bool;
      Retirar_M182 : Bool;
      Continuar_M182 : Bool;
      Entrar_M182 : Bool;
      EmiOK_M182 : Bool;
      FinLote_M183 : Bool;
      Especial_M183 : Bool;
      Bit_02_M183 : Bool;
      Retroceder_M183 : Bool;
      Retirar_M183 : Bool;
      Continuar_M183 : Bool;
      Entrar_M183 : Bool;
      EmiOK_M183 : Bool;
      FinLote_M184 : Bool;
      Especial_M184 : Bool;
      Bit_02_M184 : Bool;
      Retroceder_M184 : Bool;
      Retirar_M184 : Bool;
      Continuar_M184 : Bool;
      Entrar_M184 : Bool;
      EmiOK_M184 : Bool;
      FinLote_M185 : Bool;
      Especial_M185 : Bool;
      Bit_02_M185 : Bool;
      Retroceder_M185 : Bool;
      Retirar_M185 : Bool;
      Continuar_M185 : Bool;
      Entrar_M185 : Bool;
      EmiOK_M185 : Bool;
      FinLote_M186 : Bool;
      Especial_M186 : Bool;
      Bit_02_M186 : Bool;
      Retroceder_M186 : Bool;
      Retirar_M186 : Bool;
      Continuar_M186 : Bool;
      Entrar_M186 : Bool;
      EmiOK_M186 : Bool;
      FinLote_M187 : Bool;
      Especial_M187 : Bool;
      Bit_02_M187 : Bool;
      Retroceder_M187 : Bool;
      Retirar_M187 : Bool;
      Continuar_M187 : Bool;
      Entrar_M187 : Bool;
      EmiOK_M187 : Bool;
      FinLote_M188 : Bool;
      Especial_M188 : Bool;
      Bit_02_M188 : Bool;
      Retroceder_M188 : Bool;
      Retirar_M188 : Bool;
      Continuar_M188 : Bool;
      Entrar_M188 : Bool;
      EmiOK_M188 : Bool;
      FinLote_M189 : Bool;
      Especial_M189 : Bool;
      Bit_02_M189 : Bool;
      Retroceder_M189 : Bool;
      Retirar_M189 : Bool;
      Continuar_M189 : Bool;
      Entrar_M189 : Bool;
      EmiOK_M189 : Bool;
      FinLote_M190 : Bool;
      Especial_M190 : Bool;
      Bit_02_M190 : Bool;
      Retroceder_M190 : Bool;
      Retirar_M190 : Bool;
      Continuar_M190 : Bool;
      Entrar_M190 : Bool;
      EmiOK_M190 : Bool;
      FinLote_M191 : Bool;
      Especial_M191 : Bool;
      Bit_02_M191 : Bool;
      Retroceder_M191 : Bool;
      Retirar_M191 : Bool;
      Continuar_M191 : Bool;
      Entrar_M191 : Bool;
      EmiOK_M191 : Bool;
      FinLote_M192 : Bool;
      Especial_M192 : Bool;
      Bit_02_M192 : Bool;
      Retroceder_M192 : Bool;
      Retirar_M192 : Bool;
      Continuar_M192 : Bool;
      Entrar_M192 : Bool;
      EmiOK_M192 : Bool;
      FinLote_M193 : Bool;
      Especial_M193 : Bool;
      Bit_02_M193 : Bool;
      Retroceder_M193 : Bool;
      Retirar_M193 : Bool;
      Continuar_M193 : Bool;
      Entrar_M193 : Bool;
      EmiOK_M193 : Bool;
      FinLote_M194 : Bool;
      Especial_M194 : Bool;
      Bit_02_M194 : Bool;
      Retroceder_M194 : Bool;
      Retirar_M194 : Bool;
      Continuar_M194 : Bool;
      Entrar_M194 : Bool;
      EmiOK_M194 : Bool;
      FinLote_M195 : Bool;
      Especial_M195 : Bool;
      Bit_02_M195 : Bool;
      Retroceder_M195 : Bool;
      Retirar_M195 : Bool;
      Continuar_M195 : Bool;
      Entrar_M195 : Bool;
      EmiOK_M195 : Bool;
      FinLote_M196 : Bool;
      Especial_M196 : Bool;
      Bit_02_M196 : Bool;
      Retroceder_M196 : Bool;
      Retirar_M196 : Bool;
      Continuar_M196 : Bool;
      Entrar_M196 : Bool;
      EmiOK_M196 : Bool;
      FinLote_M197 : Bool;
      Especial_M197 : Bool;
      Bit_02_M197 : Bool;
      Retroceder_M197 : Bool;
      Retirar_M197 : Bool;
      Continuar_M197 : Bool;
      Entrar_M197 : Bool;
      EmiOK_M197 : Bool;
      FinLote_M198 : Bool;
      Especial_M198 : Bool;
      Bit_02_M198 : Bool;
      Retroceder_M198 : Bool;
      Retirar_M198 : Bool;
      Continuar_M198 : Bool;
      Entrar_M198 : Bool;
      EmiOK_M198 : Bool;
      FinLote_M199 : Bool;
      Especial_M199 : Bool;
      Bit_02_M199 : Bool;
      Retroceder_M199 : Bool;
      Retirar_M199 : Bool;
      Continuar_M199 : Bool;
      Entrar_M199 : Bool;
      EmiOK_M199 : Bool;
      FinLote_M200 : Bool;
      Especial_M200 : Bool;
      Bit_02_M200 : Bool;
      Retroceder_M200 : Bool;
      Retirar_M200 : Bool;
      Continuar_M200 : Bool;
      Entrar_M200 : Bool;
      EmiOK_M200 : Bool;
      FinLote_M201 : Bool;
      Especial_M201 : Bool;
      Bit_02_M201 : Bool;
      Retroceder_M201 : Bool;
      Retirar_M201 : Bool;
      Continuar_M201 : Bool;
      Entrar_M201 : Bool;
      EmiOK_M201 : Bool;
      FinLote_M202 : Bool;
      Especial_M202 : Bool;
      Bit_02_M202 : Bool;
      Retroceder_M202 : Bool;
      Retirar_M202 : Bool;
      Continuar_M202 : Bool;
      Entrar_M202 : Bool;
      EmiOK_M202 : Bool;
      FinLote_M203 : Bool;
      Especial_M203 : Bool;
      Bit_02_M203 : Bool;
      Retroceder_M203 : Bool;
      Retirar_M203 : Bool;
      Continuar_M203 : Bool;
      Entrar_M203 : Bool;
      EmiOK_M203 : Bool;
      FinLote_M204 : Bool;
      Especial_M204 : Bool;
      Bit_02_M204 : Bool;
      Retroceder_M204 : Bool;
      Retirar_M204 : Bool;
      Continuar_M204 : Bool;
      Entrar_M204 : Bool;
      EmiOK_M204 : Bool;
      FinLote_M205 : Bool;
      Especial_M205 : Bool;
      Bit_02_M205 : Bool;
      Retroceder_M205 : Bool;
      Retirar_M205 : Bool;
      Continuar_M205 : Bool;
      Entrar_M205 : Bool;
      EmiOK_M205 : Bool;
      FinLote_M206 : Bool;
      Especial_M206 : Bool;
      Bit_02_M206 : Bool;
      Retroceder_M206 : Bool;
      Retirar_M206 : Bool;
      Continuar_M206 : Bool;
      Entrar_M206 : Bool;
      EmiOK_M206 : Bool;
      FinLote_M207 : Bool;
      Especial_M207 : Bool;
      Bit_02_M207 : Bool;
      Retroceder_M207 : Bool;
      Retirar_M207 : Bool;
      Continuar_M207 : Bool;
      Entrar_M207 : Bool;
      EmiOK_M207 : Bool;
      FinLote_M208 : Bool;
      Especial_M208 : Bool;
      Bit_02_M208 : Bool;
      Retroceder_M208 : Bool;
      Retirar_M208 : Bool;
      Continuar_M208 : Bool;
      Entrar_M208 : Bool;
      EmiOK_M208 : Bool;
      FinLote_M209 : Bool;
      Especial_M209 : Bool;
      Bit_02_M209 : Bool;
      Retroceder_M209 : Bool;
      Retirar_M209 : Bool;
      Continuar_M209 : Bool;
      Entrar_M209 : Bool;
      EmiOK_M209 : Bool;
      FinLote_M210 : Bool;
      Especial_M210 : Bool;
      Bit_02_M210 : Bool;
      Retroceder_M210 : Bool;
      Retirar_M210 : Bool;
      Continuar_M210 : Bool;
      Entrar_M210 : Bool;
      EmiOK_M210 : Bool;
      FinLote_M211 : Bool;
      Especial_M211 : Bool;
      Bit_02_M211 : Bool;
      Retroceder_M211 : Bool;
      Retirar_M211 : Bool;
      Continuar_M211 : Bool;
      Entrar_M211 : Bool;
      EmiOK_M211 : Bool;
      FinLote_M212 : Bool;
      Especial_M212 : Bool;
      Bit_02_M212 : Bool;
      Retroceder_M212 : Bool;
      Retirar_M212 : Bool;
      Continuar_M212 : Bool;
      Entrar_M212 : Bool;
      EmiOK_M212 : Bool;
      FinLote_M213 : Bool;
      Especial_M213 : Bool;
      Bit_02_M213 : Bool;
      Retroceder_M213 : Bool;
      Retirar_M213 : Bool;
      Continuar_M213 : Bool;
      Entrar_M213 : Bool;
      EmiOK_M213 : Bool;
      FinLote_M214 : Bool;
      Especial_M214 : Bool;
      Bit_02_M214 : Bool;
      Retroceder_M214 : Bool;
      Retirar_M214 : Bool;
      Continuar_M214 : Bool;
      Entrar_M214 : Bool;
      EmiOK_M214 : Bool;
      FinLote_M215 : Bool;
      Especial_M215 : Bool;
      Bit_02_M215 : Bool;
      Retroceder_M215 : Bool;
      Retirar_M215 : Bool;
      Continuar_M215 : Bool;
      Entrar_M215 : Bool;
      EmiOK_M215 : Bool;
      FinLote_M216 : Bool;
      Especial_M216 : Bool;
      Bit_02_M216 : Bool;
      Retroceder_M216 : Bool;
      Retirar_M216 : Bool;
      Continuar_M216 : Bool;
      Entrar_M216 : Bool;
      EmiOK_M216 : Bool;
      FinLote_M217 : Bool;
      Especial_M217 : Bool;
      Bit_02_M217 : Bool;
      Retroceder_M217 : Bool;
      Retirar_M217 : Bool;
      Continuar_M217 : Bool;
      Entrar_M217 : Bool;
      EmiOK_M217 : Bool;
      FinLote_M218 : Bool;
      Especial_M218 : Bool;
      Bit_02_M218 : Bool;
      Retroceder_M218 : Bool;
      Retirar_M218 : Bool;
      Continuar_M218 : Bool;
      Entrar_M218 : Bool;
      EmiOK_M218 : Bool;
      FinLote_M219 : Bool;
      Especial_M219 : Bool;
      Bit_02_M219 : Bool;
      Retroceder_M219 : Bool;
      Retirar_M219 : Bool;
      Continuar_M219 : Bool;
      Entrar_M219 : Bool;
      EmiOK_M219 : Bool;
      FinLote_M220 : Bool;
      Especial_M220 : Bool;
      Bit_02_M220 : Bool;
      Retroceder_M220 : Bool;
      Retirar_M220 : Bool;
      Continuar_M220 : Bool;
      Entrar_M220 : Bool;
      EmiOK_M220 : Bool;
      FinLote_M221 : Bool;
      Especial_M221 : Bool;
      Bit_02_M221 : Bool;
      Retroceder_M221 : Bool;
      Retirar_M221 : Bool;
      Continuar_M221 : Bool;
      Entrar_M221 : Bool;
      EmiOK_M221 : Bool;
      FinLote_M222 : Bool;
      Especial_M222 : Bool;
      Bit_02_M222 : Bool;
      Retroceder_M222 : Bool;
      Retirar_M222 : Bool;
      Continuar_M222 : Bool;
      Entrar_M222 : Bool;
      EmiOK_M222 : Bool;
      FinLote_M223 : Bool;
      Especial_M223 : Bool;
      Bit_02_M223 : Bool;
      Retroceder_M223 : Bool;
      Retirar_M223 : Bool;
      Continuar_M223 : Bool;
      Entrar_M223 : Bool;
      EmiOK_M223 : Bool;
      FinLote_M224 : Bool;
      Especial_M224 : Bool;
      Bit_02_M224 : Bool;
      Retroceder_M224 : Bool;
      Retirar_M224 : Bool;
      Continuar_M224 : Bool;
      Entrar_M224 : Bool;
      EmiOK_M224 : Bool;
      FinLote_M225 : Bool;
      Especial_M225 : Bool;
      Bit_02_M225 : Bool;
      Retroceder_M225 : Bool;
      Retirar_M225 : Bool;
      Continuar_M225 : Bool;
      Entrar_M225 : Bool;
      EmiOK_M225 : Bool;
      FinLote_M226 : Bool;
      Especial_M226 : Bool;
      Bit_02_M226 : Bool;
      Retroceder_M226 : Bool;
      Retirar_M226 : Bool;
      Continuar_M226 : Bool;
      Entrar_M226 : Bool;
      EmiOK_M226 : Bool;
      FinLote_M227 : Bool;
      Especial_M227 : Bool;
      Bit_02_M227 : Bool;
      Retroceder_M227 : Bool;
      Retirar_M227 : Bool;
      Continuar_M227 : Bool;
      Entrar_M227 : Bool;
      EmiOK_M227 : Bool;
      FinLote_M228 : Bool;
      Especial_M228 : Bool;
      Bit_02_M228 : Bool;
      Retroceder_M228 : Bool;
      Retirar_M228 : Bool;
      Continuar_M228 : Bool;
      Entrar_M228 : Bool;
      EmiOK_M228 : Bool;
      FinLote_M229 : Bool;
      Especial_M229 : Bool;
      Bit_02_M229 : Bool;
      Retroceder_M229 : Bool;
      Retirar_M229 : Bool;
      Continuar_M229 : Bool;
      Entrar_M229 : Bool;
      EmiOK_M229 : Bool;
      FinLote_M230 : Bool;
      Especial_M230 : Bool;
      Bit_02_M230 : Bool;
      Retroceder_M230 : Bool;
      Retirar_M230 : Bool;
      Continuar_M230 : Bool;
      Entrar_M230 : Bool;
      EmiOK_M230 : Bool;
      FinLote_M231 : Bool;
      Especial_M231 : Bool;
      Bit_02_M231 : Bool;
      Retroceder_M231 : Bool;
      Retirar_M231 : Bool;
      Continuar_M231 : Bool;
      Entrar_M231 : Bool;
      EmiOK_M231 : Bool;
      FinLote_M232 : Bool;
      Especial_M232 : Bool;
      Bit_02_M232 : Bool;
      Retroceder_M232 : Bool;
      Retirar_M232 : Bool;
      Continuar_M232 : Bool;
      Entrar_M232 : Bool;
      EmiOK_M232 : Bool;
      FinLote_M233 : Bool;
      Especial_M233 : Bool;
      Bit_02_M233 : Bool;
      Retroceder_M233 : Bool;
      Retirar_M233 : Bool;
      Continuar_M233 : Bool;
      Entrar_M233 : Bool;
      EmiOK_M233 : Bool;
      FinLote_M234 : Bool;
      Especial_M234 : Bool;
      Bit_02_M234 : Bool;
      Retroceder_M234 : Bool;
      Retirar_M234 : Bool;
      Continuar_M234 : Bool;
      Entrar_M234 : Bool;
      EmiOK_M234 : Bool;
      FinLote_M235 : Bool;
      Especial_M235 : Bool;
      Bit_02_M235 : Bool;
      Retroceder_M235 : Bool;
      Retirar_M235 : Bool;
      Continuar_M235 : Bool;
      Entrar_M235 : Bool;
      EmiOK_M235 : Bool;
      FinLote_M236 : Bool;
      Especial_M236 : Bool;
      Bit_02_M236 : Bool;
      Retroceder_M236 : Bool;
      Retirar_M236 : Bool;
      Continuar_M236 : Bool;
      Entrar_M236 : Bool;
      EmiOK_M236 : Bool;
      FinLote_M237 : Bool;
      Especial_M237 : Bool;
      Bit_02_M237 : Bool;
      Retroceder_M237 : Bool;
      Retirar_M237 : Bool;
      Continuar_M237 : Bool;
      Entrar_M237 : Bool;
      EmiOK_M237 : Bool;
      FinLote_M238 : Bool;
      Especial_M238 : Bool;
      Bit_02_M238 : Bool;
      Retroceder_M238 : Bool;
      Retirar_M238 : Bool;
      Continuar_M238 : Bool;
      Entrar_M238 : Bool;
      EmiOK_M238 : Bool;
      FinLote_M239 : Bool;
      Especial_M239 : Bool;
      Bit_02_M239 : Bool;
      Retroceder_M239 : Bool;
      Retirar_M239 : Bool;
      Continuar_M239 : Bool;
      Entrar_M239 : Bool;
      EmiOK_M239 : Bool;
      FinLote_M240 : Bool;
      Especial_M240 : Bool;
      Bit_02_M240 : Bool;
      Retroceder_M240 : Bool;
      Retirar_M240 : Bool;
      Continuar_M240 : Bool;
      Entrar_M240 : Bool;
      EmiOK_M240 : Bool;
      FinLote_M241 : Bool;
      Especial_M241 : Bool;
      Bit_02_M241 : Bool;
      Retroceder_M241 : Bool;
      Retirar_M241 : Bool;
      Continuar_M241 : Bool;
      Entrar_M241 : Bool;
      EmiOK_M241 : Bool;
      FinLote_M242 : Bool;
      Especial_M242 : Bool;
      Bit_02_M242 : Bool;
      Retroceder_M242 : Bool;
      Retirar_M242 : Bool;
      Continuar_M242 : Bool;
      Entrar_M242 : Bool;
      EmiOK_M242 : Bool;
      FinLote_M243 : Bool;
      Especial_M243 : Bool;
      Bit_02_M243 : Bool;
      Retroceder_M243 : Bool;
      Retirar_M243 : Bool;
      Continuar_M243 : Bool;
      Entrar_M243 : Bool;
      EmiOK_M243 : Bool;
      FinLote_M244 : Bool;
      Especial_M244 : Bool;
      Bit_02_M244 : Bool;
      Retroceder_M244 : Bool;
      Retirar_M244 : Bool;
      Continuar_M244 : Bool;
      Entrar_M244 : Bool;
      EmiOK_M244 : Bool;
      FinLote_M245 : Bool;
      Especial_M245 : Bool;
      Bit_02_M245 : Bool;
      Retroceder_M245 : Bool;
      Retirar_M245 : Bool;
      Continuar_M245 : Bool;
      Entrar_M245 : Bool;
      EmiOK_M245 : Bool;
      FinLote_M246 : Bool;
      Especial_M246 : Bool;
      Bit_02_M246 : Bool;
      Retroceder_M246 : Bool;
      Retirar_M246 : Bool;
      Continuar_M246 : Bool;
      Entrar_M246 : Bool;
      EmiOK_M246 : Bool;
      FinLote_M247 : Bool;
      Especial_M247 : Bool;
      Bit_02_M247 : Bool;
      Retroceder_M247 : Bool;
      Retirar_M247 : Bool;
      Continuar_M247 : Bool;
      Entrar_M247 : Bool;
      EmiOK_M247 : Bool;
      FinLote_M248 : Bool;
      Especial_M248 : Bool;
      Bit_02_M248 : Bool;
      Retroceder_M248 : Bool;
      Retirar_M248 : Bool;
      Continuar_M248 : Bool;
      Entrar_M248 : Bool;
      EmiOK_M248 : Bool;
      FinLote_M249 : Bool;
      Especial_M249 : Bool;
      Bit_02_M249 : Bool;
      Retroceder_M249 : Bool;
      Retirar_M249 : Bool;
      Continuar_M249 : Bool;
      Entrar_M249 : Bool;
      EmiOK_M249 : Bool;
      FinLote_M250 : Bool;
      Especial_M250 : Bool;
      Bit_02_M250 : Bool;
      Retroceder_M250 : Bool;
      Retirar_M250 : Bool;
      Continuar_M250 : Bool;
      Entrar_M250 : Bool;
      EmiOK_M250 : Bool;
      FinLote_M251 : Bool;
      Especial_M251 : Bool;
      Bit_02_M251 : Bool;
      Retroceder_M251 : Bool;
      Retirar_M251 : Bool;
      Continuar_M251 : Bool;
      Entrar_M251 : Bool;
      EmiOK_M251 : Bool;
      FinLote_M252 : Bool;
      Especial_M252 : Bool;
      Bit_02_M252 : Bool;
      Retroceder_M252 : Bool;
      Retirar_M252 : Bool;
      Continuar_M252 : Bool;
      Entrar_M252 : Bool;
      EmiOK_M252 : Bool;
      FinLote_M253 : Bool;
      Especial_M253 : Bool;
      Bit_02_M253 : Bool;
      Retroceder_M253 : Bool;
      Retirar_M253 : Bool;
      Continuar_M253 : Bool;
      Entrar_M253 : Bool;
      EmiOK_M253 : Bool;
      FinLote_M254 : Bool;
      Especial_M254 : Bool;
      Bit_02_M254 : Bool;
      Retroceder_M254 : Bool;
      Retirar_M254 : Bool;
      Continuar_M254 : Bool;
      Entrar_M254 : Bool;
      EmiOK_M254 : Bool;
      FinLote_M255 : Bool;
      Especial_M255 : Bool;
      Bit_02_M255 : Bool;
      Retroceder_M255 : Bool;
      Retirar_M255 : Bool;
      Continuar_M255 : Bool;
      Entrar_M255 : Bool;
      EmiOK_M255 : Bool;
      FinLote_M256 : Bool;
      Especial_M256 : Bool;
      Bit_02_M256 : Bool;
      Retroceder_M256 : Bool;
      Retirar_M256 : Bool;
      Continuar_M256 : Bool;
      Entrar_M256 : Bool;
      EmiOK_M256 : Bool;
      FinLote_M257 : Bool;
      Especial_M257 : Bool;
      Bit_02_M257 : Bool;
      Retroceder_M257 : Bool;
      Retirar_M257 : Bool;
      Continuar_M257 : Bool;
      Entrar_M257 : Bool;
      EmiOK_M257 : Bool;
      FinLote_M258 : Bool;
      Especial_M258 : Bool;
      Bit_02_M258 : Bool;
      Retroceder_M258 : Bool;
      Retirar_M258 : Bool;
      Continuar_M258 : Bool;
      Entrar_M258 : Bool;
      EmiOK_M258 : Bool;
      FinLote_M259 : Bool;
      Especial_M259 : Bool;
      Bit_02_M259 : Bool;
      Retroceder_M259 : Bool;
      Retirar_M259 : Bool;
      Continuar_M259 : Bool;
      Entrar_M259 : Bool;
      EmiOK_M259 : Bool;
      FinLote_M260 : Bool;
      Especial_M260 : Bool;
      Bit_02_M260 : Bool;
      Retroceder_M260 : Bool;
      Retirar_M260 : Bool;
      Continuar_M260 : Bool;
      Entrar_M260 : Bool;
      EmiOK_M260 : Bool;
      FinLote_M261 : Bool;
      Especial_M261 : Bool;
      Bit_02_M261 : Bool;
      Retroceder_M261 : Bool;
      Retirar_M261 : Bool;
      Continuar_M261 : Bool;
      Entrar_M261 : Bool;
      EmiOK_M261 : Bool;
      FinLote_M262 : Bool;
      Especial_M262 : Bool;
      Bit_02_M262 : Bool;
      Retroceder_M262 : Bool;
      Retirar_M262 : Bool;
      Continuar_M262 : Bool;
      Entrar_M262 : Bool;
      EmiOK_M262 : Bool;
      FinLote_M263 : Bool;
      Especial_M263 : Bool;
      Bit_02_M263 : Bool;
      Retroceder_M263 : Bool;
      Retirar_M263 : Bool;
      Continuar_M263 : Bool;
      Entrar_M263 : Bool;
      EmiOK_M263 : Bool;
      FinLote_M264 : Bool;
      Especial_M264 : Bool;
      Bit_02_M264 : Bool;
      Retroceder_M264 : Bool;
      Retirar_M264 : Bool;
      Continuar_M264 : Bool;
      Entrar_M264 : Bool;
      EmiOK_M264 : Bool;
      FinLote_M265 : Bool;
      Especial_M265 : Bool;
      Bit_02_M265 : Bool;
      Retroceder_M265 : Bool;
      Retirar_M265 : Bool;
      Continuar_M265 : Bool;
      Entrar_M265 : Bool;
      EmiOK_M265 : Bool;
      FinLote_M266 : Bool;
      Especial_M266 : Bool;
      Bit_02_M266 : Bool;
      Retroceder_M266 : Bool;
      Retirar_M266 : Bool;
      Continuar_M266 : Bool;
      Entrar_M266 : Bool;
      EmiOK_M266 : Bool;
      FinLote_M267 : Bool;
      Especial_M267 : Bool;
      Bit_02_M267 : Bool;
      Retroceder_M267 : Bool;
      Retirar_M267 : Bool;
      Continuar_M267 : Bool;
      Entrar_M267 : Bool;
      EmiOK_M267 : Bool;
      FinLote_M268 : Bool;
      Especial_M268 : Bool;
      Bit_02_M268 : Bool;
      Retroceder_M268 : Bool;
      Retirar_M268 : Bool;
      Continuar_M268 : Bool;
      Entrar_M268 : Bool;
      EmiOK_M268 : Bool;
      FinLote_M269 : Bool;
      Especial_M269 : Bool;
      Bit_02_M269 : Bool;
      Retroceder_M269 : Bool;
      Retirar_M269 : Bool;
      Continuar_M269 : Bool;
      Entrar_M269 : Bool;
      EmiOK_M269 : Bool;
      FinLote_M270 : Bool;
      Especial_M270 : Bool;
      Bit_02_M270 : Bool;
      Retroceder_M270 : Bool;
      Retirar_M270 : Bool;
      Continuar_M270 : Bool;
      Entrar_M270 : Bool;
      EmiOK_M270 : Bool;
      FinLote_M271 : Bool;
      Especial_M271 : Bool;
      Bit_02_M271 : Bool;
      Retroceder_M271 : Bool;
      Retirar_M271 : Bool;
      Continuar_M271 : Bool;
      Entrar_M271 : Bool;
      EmiOK_M271 : Bool;
      FinLote_M272 : Bool;
      Especial_M272 : Bool;
      Bit_02_M272 : Bool;
      Retroceder_M272 : Bool;
      Retirar_M272 : Bool;
      Continuar_M272 : Bool;
      Entrar_M272 : Bool;
      EmiOK_M272 : Bool;
      FinLote_M273 : Bool;
      Especial_M273 : Bool;
      Bit_02_M273 : Bool;
      Retroceder_M273 : Bool;
      Retirar_M273 : Bool;
      Continuar_M273 : Bool;
      Entrar_M273 : Bool;
      EmiOK_M273 : Bool;
      FinLote_M274 : Bool;
      Especial_M274 : Bool;
      Bit_02_M274 : Bool;
      Retroceder_M274 : Bool;
      Retirar_M274 : Bool;
      Continuar_M274 : Bool;
      Entrar_M274 : Bool;
      EmiOK_M274 : Bool;
      FinLote_M275 : Bool;
      Especial_M275 : Bool;
      Bit_02_M275 : Bool;
      Retroceder_M275 : Bool;
      Retirar_M275 : Bool;
      Continuar_M275 : Bool;
      Entrar_M275 : Bool;
      EmiOK_M275 : Bool;
      FinLote_M276 : Bool;
      Especial_M276 : Bool;
      Bit_02_M276 : Bool;
      Retroceder_M276 : Bool;
      Retirar_M276 : Bool;
      Continuar_M276 : Bool;
      Entrar_M276 : Bool;
      EmiOK_M276 : Bool;
      FinLote_M277 : Bool;
      Especial_M277 : Bool;
      Bit_02_M277 : Bool;
      Retroceder_M277 : Bool;
      Retirar_M277 : Bool;
      Continuar_M277 : Bool;
      Entrar_M277 : Bool;
      EmiOK_M277 : Bool;
      FinLote_M278 : Bool;
      Especial_M278 : Bool;
      Bit_02_M278 : Bool;
      Retroceder_M278 : Bool;
      Retirar_M278 : Bool;
      Continuar_M278 : Bool;
      Entrar_M278 : Bool;
      EmiOK_M278 : Bool;
      FinLote_M279 : Bool;
      Especial_M279 : Bool;
      Bit_02_M279 : Bool;
      Retroceder_M279 : Bool;
      Retirar_M279 : Bool;
      Continuar_M279 : Bool;
      Entrar_M279 : Bool;
      EmiOK_M279 : Bool;
      FinLote_M280 : Bool;
      Especial_M280 : Bool;
      Bit_02_M280 : Bool;
      Retroceder_M280 : Bool;
      Retirar_M280 : Bool;
      Continuar_M280 : Bool;
      Entrar_M280 : Bool;
      EmiOK_M280 : Bool;
      FinLote_M281 : Bool;
      Especial_M281 : Bool;
      Bit_02_M281 : Bool;
      Retroceder_M281 : Bool;
      Retirar_M281 : Bool;
      Continuar_M281 : Bool;
      Entrar_M281 : Bool;
      EmiOK_M281 : Bool;
      FinLote_M282 : Bool;
      Especial_M282 : Bool;
      Bit_02_M282 : Bool;
      Retroceder_M282 : Bool;
      Retirar_M282 : Bool;
      Continuar_M282 : Bool;
      Entrar_M282 : Bool;
      EmiOK_M282 : Bool;
      FinLote_M283 : Bool;
      Especial_M283 : Bool;
      Bit_02_M283 : Bool;
      Retroceder_M283 : Bool;
      Retirar_M283 : Bool;
      Continuar_M283 : Bool;
      Entrar_M283 : Bool;
      EmiOK_M283 : Bool;
      FinLote_M284 : Bool;
      Especial_M284 : Bool;
      Bit_02_M284 : Bool;
      Retroceder_M284 : Bool;
      Retirar_M284 : Bool;
      Continuar_M284 : Bool;
      Entrar_M284 : Bool;
      EmiOK_M284 : Bool;
      FinLote_M285 : Bool;
      Especial_M285 : Bool;
      Bit_02_M285 : Bool;
      Retroceder_M285 : Bool;
      Retirar_M285 : Bool;
      Continuar_M285 : Bool;
      Entrar_M285 : Bool;
      EmiOK_M285 : Bool;
      FinLote_M286 : Bool;
      Especial_M286 : Bool;
      Bit_02_M286 : Bool;
      Retroceder_M286 : Bool;
      Retirar_M286 : Bool;
      Continuar_M286 : Bool;
      Entrar_M286 : Bool;
      EmiOK_M286 : Bool;
      FinLote_M287 : Bool;
      Especial_M287 : Bool;
      Bit_02_M287 : Bool;
      Retroceder_M287 : Bool;
      Retirar_M287 : Bool;
      Continuar_M287 : Bool;
      Entrar_M287 : Bool;
      EmiOK_M287 : Bool;
      FinLote_M288 : Bool;
      Especial_M288 : Bool;
      Bit_02_M288 : Bool;
      Retroceder_M288 : Bool;
      Retirar_M288 : Bool;
      Continuar_M288 : Bool;
      Entrar_M288 : Bool;
      EmiOK_M288 : Bool;
      FinLote_M289 : Bool;
      Especial_M289 : Bool;
      Bit_02_M289 : Bool;
      Retroceder_M289 : Bool;
      Retirar_M289 : Bool;
      Continuar_M289 : Bool;
      Entrar_M289 : Bool;
      EmiOK_M289 : Bool;
      FinLote_M290 : Bool;
      Especial_M290 : Bool;
      Bit_02_M290 : Bool;
      Retroceder_M290 : Bool;
      Retirar_M290 : Bool;
      Continuar_M290 : Bool;
      Entrar_M290 : Bool;
      EmiOK_M290 : Bool;
      FinLote_M291 : Bool;
      Especial_M291 : Bool;
      Bit_02_M291 : Bool;
      Retroceder_M291 : Bool;
      Retirar_M291 : Bool;
      Continuar_M291 : Bool;
      Entrar_M291 : Bool;
      EmiOK_M291 : Bool;
      FinLote_M292 : Bool;
      Especial_M292 : Bool;
      Bit_02_M292 : Bool;
      Retroceder_M292 : Bool;
      Retirar_M292 : Bool;
      Continuar_M292 : Bool;
      Entrar_M292 : Bool;
      EmiOK_M292 : Bool;
      FinLote_M293 : Bool;
      Especial_M293 : Bool;
      Bit_02_M293 : Bool;
      Retroceder_M293 : Bool;
      Retirar_M293 : Bool;
      Continuar_M293 : Bool;
      Entrar_M293 : Bool;
      EmiOK_M293 : Bool;
      FinLote_M294 : Bool;
      Especial_M294 : Bool;
      Bit_02_M294 : Bool;
      Retroceder_M294 : Bool;
      Retirar_M294 : Bool;
      Continuar_M294 : Bool;
      Entrar_M294 : Bool;
      EmiOK_M294 : Bool;
      FinLote_M295 : Bool;
      Especial_M295 : Bool;
      Bit_02_M295 : Bool;
      Retroceder_M295 : Bool;
      Retirar_M295 : Bool;
      Continuar_M295 : Bool;
      Entrar_M295 : Bool;
      EmiOK_M295 : Bool;
      FinLote_M296 : Bool;
      Especial_M296 : Bool;
      Bit_02_M296 : Bool;
      Retroceder_M296 : Bool;
      Retirar_M296 : Bool;
      Continuar_M296 : Bool;
      Entrar_M296 : Bool;
      EmiOK_M296 : Bool;
      FinLote_M297 : Bool;
      Especial_M297 : Bool;
      Bit_02_M297 : Bool;
      Retroceder_M297 : Bool;
      Retirar_M297 : Bool;
      Continuar_M297 : Bool;
      Entrar_M297 : Bool;
      EmiOK_M297 : Bool;
      FinLote_M298 : Bool;
      Especial_M298 : Bool;
      Bit_02_M298 : Bool;
      Retroceder_M298 : Bool;
      Retirar_M298 : Bool;
      Continuar_M298 : Bool;
      Entrar_M298 : Bool;
      EmiOK_M298 : Bool;
      FinLote_M299 : Bool;
      Especial_M299 : Bool;
      Bit_02_M299 : Bool;
      Retroceder_M299 : Bool;
      Retirar_M299 : Bool;
      Continuar_M299 : Bool;
      Entrar_M299 : Bool;
      EmiOK_M299 : Bool;
      FinLote_M300 : Bool;
      Especial_M300 : Bool;
      Bit_02_M300 : Bool;
      Retroceder_M300 : Bool;
      Retirar_M300 : Bool;
      Continuar_M300 : Bool;
      Entrar_M300 : Bool;
      EmiOK_M300 : Bool;
      FinLote_M301 : Bool;
      Especial_M301 : Bool;
      Bit_02_M301 : Bool;
      Retroceder_M301 : Bool;
      Retirar_M301 : Bool;
      Continuar_M301 : Bool;
      Entrar_M301 : Bool;
      EmiOK_M301 : Bool;
      FinLote_M302 : Bool;
      Especial_M302 : Bool;
      Bit_02_M302 : Bool;
      Retroceder_M302 : Bool;
      Retirar_M302 : Bool;
      Continuar_M302 : Bool;
      Entrar_M302 : Bool;
      EmiOK_M302 : Bool;
      FinLote_M303 : Bool;
      Especial_M303 : Bool;
      Bit_02_M303 : Bool;
      Retroceder_M303 : Bool;
      Retirar_M303 : Bool;
      Continuar_M303 : Bool;
      Entrar_M303 : Bool;
      EmiOK_M303 : Bool;
      FinLote_M304 : Bool;
      Especial_M304 : Bool;
      Bit_02_M304 : Bool;
      Retroceder_M304 : Bool;
      Retirar_M304 : Bool;
      Continuar_M304 : Bool;
      Entrar_M304 : Bool;
      EmiOK_M304 : Bool;
      FinLote_M305 : Bool;
      Especial_M305 : Bool;
      Bit_02_M305 : Bool;
      Retroceder_M305 : Bool;
      Retirar_M305 : Bool;
      Continuar_M305 : Bool;
      Entrar_M305 : Bool;
      EmiOK_M305 : Bool;
      FinLote_M306 : Bool;
      Especial_M306 : Bool;
      Bit_02_M306 : Bool;
      Retroceder_M306 : Bool;
      Retirar_M306 : Bool;
      Continuar_M306 : Bool;
      Entrar_M306 : Bool;
      EmiOK_M306 : Bool;
      FinLote_M307 : Bool;
      Especial_M307 : Bool;
      Bit_02_M307 : Bool;
      Retroceder_M307 : Bool;
      Retirar_M307 : Bool;
      Continuar_M307 : Bool;
      Entrar_M307 : Bool;
      EmiOK_M307 : Bool;
      FinLote_M308 : Bool;
      Especial_M308 : Bool;
      Bit_02_M308 : Bool;
      Retroceder_M308 : Bool;
      Retirar_M308 : Bool;
      Continuar_M308 : Bool;
      Entrar_M308 : Bool;
      EmiOK_M308 : Bool;
      FinLote_M309 : Bool;
      Especial_M309 : Bool;
      Bit_02_M309 : Bool;
      Retroceder_M309 : Bool;
      Retirar_M309 : Bool;
      Continuar_M309 : Bool;
      Entrar_M309 : Bool;
      EmiOK_M309 : Bool;
      FinLote_M310 : Bool;
      Especial_M310 : Bool;
      Bit_02_M310 : Bool;
      Retroceder_M310 : Bool;
      Retirar_M310 : Bool;
      Continuar_M310 : Bool;
      Entrar_M310 : Bool;
      EmiOK_M310 : Bool;
      FinLote_M311 : Bool;
      Especial_M311 : Bool;
      Bit_02_M311 : Bool;
      Retroceder_M311 : Bool;
      Retirar_M311 : Bool;
      Continuar_M311 : Bool;
      Entrar_M311 : Bool;
      EmiOK_M311 : Bool;
      FinLote_M312 : Bool;
      Especial_M312 : Bool;
      Bit_02_M312 : Bool;
      Retroceder_M312 : Bool;
      Retirar_M312 : Bool;
      Continuar_M312 : Bool;
      Entrar_M312 : Bool;
      EmiOK_M312 : Bool;
      FinLote_M313 : Bool;
      Especial_M313 : Bool;
      Bit_02_M313 : Bool;
      Retroceder_M313 : Bool;
      Retirar_M313 : Bool;
      Continuar_M313 : Bool;
      Entrar_M313 : Bool;
      EmiOK_M313 : Bool;
      FinLote_M314 : Bool;
      Especial_M314 : Bool;
      Bit_02_M314 : Bool;
      Retroceder_M314 : Bool;
      Retirar_M314 : Bool;
      Continuar_M314 : Bool;
      Entrar_M314 : Bool;
      EmiOK_M314 : Bool;
      FinLote_M315 : Bool;
      Especial_M315 : Bool;
      Bit_02_M315 : Bool;
      Retroceder_M315 : Bool;
      Retirar_M315 : Bool;
      Continuar_M315 : Bool;
      Entrar_M315 : Bool;
      EmiOK_M315 : Bool;
      FinLote_M316 : Bool;
      Especial_M316 : Bool;
      Bit_02_M316 : Bool;
      Retroceder_M316 : Bool;
      Retirar_M316 : Bool;
      Continuar_M316 : Bool;
      Entrar_M316 : Bool;
      EmiOK_M316 : Bool;
      FinLote_M317 : Bool;
      Especial_M317 : Bool;
      Bit_02_M317 : Bool;
      Retroceder_M317 : Bool;
      Retirar_M317 : Bool;
      Continuar_M317 : Bool;
      Entrar_M317 : Bool;
      EmiOK_M317 : Bool;
      FinLote_M318 : Bool;
      Especial_M318 : Bool;
      Bit_02_M318 : Bool;
      Retroceder_M318 : Bool;
      Retirar_M318 : Bool;
      Continuar_M318 : Bool;
      Entrar_M318 : Bool;
      EmiOK_M318 : Bool;
      FinLote_M319 : Bool;
      Especial_M319 : Bool;
      Bit_02_M319 : Bool;
      Retroceder_M319 : Bool;
      Retirar_M319 : Bool;
      Continuar_M319 : Bool;
      Entrar_M319 : Bool;
      EmiOK_M319 : Bool;
      FinLote_M320 : Bool;
      Especial_M320 : Bool;
      Bit_02_M320 : Bool;
      Retroceder_M320 : Bool;
      Retirar_M320 : Bool;
      Continuar_M320 : Bool;
      Entrar_M320 : Bool;
      EmiOK_M320 : Bool;
      FinLote_M321 : Bool;
      Especial_M321 : Bool;
      Bit_02_M321 : Bool;
      Retroceder_M321 : Bool;
      Retirar_M321 : Bool;
      Continuar_M321 : Bool;
      Entrar_M321 : Bool;
      EmiOK_M321 : Bool;
      FinLote_M322 : Bool;
      Especial_M322 : Bool;
      Bit_02_M322 : Bool;
      Retroceder_M322 : Bool;
      Retirar_M322 : Bool;
      Continuar_M322 : Bool;
      Entrar_M322 : Bool;
      EmiOK_M322 : Bool;
      FinLote_M323 : Bool;
      Especial_M323 : Bool;
      Bit_02_M323 : Bool;
      Retroceder_M323 : Bool;
      Retirar_M323 : Bool;
      Continuar_M323 : Bool;
      Entrar_M323 : Bool;
      EmiOK_M323 : Bool;
      FinLote_M324 : Bool;
      Especial_M324 : Bool;
      Bit_02_M324 : Bool;
      Retroceder_M324 : Bool;
      Retirar_M324 : Bool;
      Continuar_M324 : Bool;
      Entrar_M324 : Bool;
      EmiOK_M324 : Bool;
      FinLote_M325 : Bool;
      Especial_M325 : Bool;
      Bit_02_M325 : Bool;
      Retroceder_M325 : Bool;
      Retirar_M325 : Bool;
      Continuar_M325 : Bool;
      Entrar_M325 : Bool;
      EmiOK_M325 : Bool;
      FinLote_M326 : Bool;
      Especial_M326 : Bool;
      Bit_02_M326 : Bool;
      Retroceder_M326 : Bool;
      Retirar_M326 : Bool;
      Continuar_M326 : Bool;
      Entrar_M326 : Bool;
      EmiOK_M326 : Bool;
      FinLote_M327 : Bool;
      Especial_M327 : Bool;
      Bit_02_M327 : Bool;
      Retroceder_M327 : Bool;
      Retirar_M327 : Bool;
      Continuar_M327 : Bool;
      Entrar_M327 : Bool;
      EmiOK_M327 : Bool;
      FinLote_M328 : Bool;
      Especial_M328 : Bool;
      Bit_02_M328 : Bool;
      Retroceder_M328 : Bool;
      Retirar_M328 : Bool;
      Continuar_M328 : Bool;
      Entrar_M328 : Bool;
      EmiOK_M328 : Bool;
      FinLote_M329 : Bool;
      Especial_M329 : Bool;
      Bit_02_M329 : Bool;
      Retroceder_M329 : Bool;
      Retirar_M329 : Bool;
      Continuar_M329 : Bool;
      Entrar_M329 : Bool;
      EmiOK_M329 : Bool;
      FinLote_M330 : Bool;
      Especial_M330 : Bool;
      Bit_02_M330 : Bool;
      Retroceder_M330 : Bool;
      Retirar_M330 : Bool;
      Continuar_M330 : Bool;
      Entrar_M330 : Bool;
      EmiOK_M330 : Bool;
      FinLote_M331 : Bool;
      Especial_M331 : Bool;
      Bit_02_M331 : Bool;
      Retroceder_M331 : Bool;
      Retirar_M331 : Bool;
      Continuar_M331 : Bool;
      Entrar_M331 : Bool;
      EmiOK_M331 : Bool;
      FinLote_M332 : Bool;
      Especial_M332 : Bool;
      Bit_02_M332 : Bool;
      Retroceder_M332 : Bool;
      Retirar_M332 : Bool;
      Continuar_M332 : Bool;
      Entrar_M332 : Bool;
      EmiOK_M332 : Bool;
      FinLote_M333 : Bool;
      Especial_M333 : Bool;
      Bit_02_M333 : Bool;
      Retroceder_M333 : Bool;
      Retirar_M333 : Bool;
      Continuar_M333 : Bool;
      Entrar_M333 : Bool;
      EmiOK_M333 : Bool;
      FinLote_M334 : Bool;
      Especial_M334 : Bool;
      Bit_02_M334 : Bool;
      Retroceder_M334 : Bool;
      Retirar_M334 : Bool;
      Continuar_M334 : Bool;
      Entrar_M334 : Bool;
      EmiOK_M334 : Bool;
      FinLote_M335 : Bool;
      Especial_M335 : Bool;
      Bit_02_M335 : Bool;
      Retroceder_M335 : Bool;
      Retirar_M335 : Bool;
      Continuar_M335 : Bool;
      Entrar_M335 : Bool;
      EmiOK_M335 : Bool;
      FinLote_M336 : Bool;
      Especial_M336 : Bool;
      Bit_02_M336 : Bool;
      Retroceder_M336 : Bool;
      Retirar_M336 : Bool;
      Continuar_M336 : Bool;
      Entrar_M336 : Bool;
      EmiOK_M336 : Bool;
      FinLote_M337 : Bool;
      Especial_M337 : Bool;
      Bit_02_M337 : Bool;
      Retroceder_M337 : Bool;
      Retirar_M337 : Bool;
      Continuar_M337 : Bool;
      Entrar_M337 : Bool;
      EmiOK_M337 : Bool;
      FinLote_M338 : Bool;
      Especial_M338 : Bool;
      Bit_02_M338 : Bool;
      Retroceder_M338 : Bool;
      Retirar_M338 : Bool;
      Continuar_M338 : Bool;
      Entrar_M338 : Bool;
      EmiOK_M338 : Bool;
      FinLote_M339 : Bool;
      Especial_M339 : Bool;
      Bit_02_M339 : Bool;
      Retroceder_M339 : Bool;
      Retirar_M339 : Bool;
      Continuar_M339 : Bool;
      Entrar_M339 : Bool;
      EmiOK_M339 : Bool;
      FinLote_M340 : Bool;
      Especial_M340 : Bool;
      Bit_02_M340 : Bool;
      Retroceder_M340 : Bool;
      Retirar_M340 : Bool;
      Continuar_M340 : Bool;
      Entrar_M340 : Bool;
      EmiOK_M340 : Bool;
      FinLote_M341 : Bool;
      Especial_M341 : Bool;
      Bit_02_M341 : Bool;
      Retroceder_M341 : Bool;
      Retirar_M341 : Bool;
      Continuar_M341 : Bool;
      Entrar_M341 : Bool;
      EmiOK_M341 : Bool;
      FinLote_M342 : Bool;
      Especial_M342 : Bool;
      Bit_02_M342 : Bool;
      Retroceder_M342 : Bool;
      Retirar_M342 : Bool;
      Continuar_M342 : Bool;
      Entrar_M342 : Bool;
      EmiOK_M342 : Bool;
      FinLote_M343 : Bool;
      Especial_M343 : Bool;
      Bit_02_M343 : Bool;
      Retroceder_M343 : Bool;
      Retirar_M343 : Bool;
      Continuar_M343 : Bool;
      Entrar_M343 : Bool;
      EmiOK_M343 : Bool;
      FinLote_M344 : Bool;
      Especial_M344 : Bool;
      Bit_02_M344 : Bool;
      Retroceder_M344 : Bool;
      Retirar_M344 : Bool;
      Continuar_M344 : Bool;
      Entrar_M344 : Bool;
      EmiOK_M344 : Bool;
      FinLote_M345 : Bool;
      Especial_M345 : Bool;
      Bit_02_M345 : Bool;
      Retroceder_M345 : Bool;
      Retirar_M345 : Bool;
      Continuar_M345 : Bool;
      Entrar_M345 : Bool;
      EmiOK_M345 : Bool;
      FinLote_M346 : Bool;
      Especial_M346 : Bool;
      Bit_02_M346 : Bool;
      Retroceder_M346 : Bool;
      Retirar_M346 : Bool;
      Continuar_M346 : Bool;
      Entrar_M346 : Bool;
      EmiOK_M346 : Bool;
      FinLote_M347 : Bool;
      Especial_M347 : Bool;
      Bit_02_M347 : Bool;
      Retroceder_M347 : Bool;
      Retirar_M347 : Bool;
      Continuar_M347 : Bool;
      Entrar_M347 : Bool;
      EmiOK_M347 : Bool;
      FinLote_M348 : Bool;
      Especial_M348 : Bool;
      Bit_02_M348 : Bool;
      Retroceder_M348 : Bool;
      Retirar_M348 : Bool;
      Continuar_M348 : Bool;
      Entrar_M348 : Bool;
      EmiOK_M348 : Bool;
      FinLote_M349 : Bool;
      Especial_M349 : Bool;
      Bit_02_M349 : Bool;
      Retroceder_M349 : Bool;
      Retirar_M349 : Bool;
      Continuar_M349 : Bool;
      Entrar_M349 : Bool;
      EmiOK_M349 : Bool;
      FinLote_M350 : Bool;
      Especial_M350 : Bool;
      Bit_02_M350 : Bool;
      Retroceder_M350 : Bool;
      Retirar_M350 : Bool;
      Continuar_M350 : Bool;
      Entrar_M350 : Bool;
      EmiOK_M350 : Bool;
      FinLote_M351 : Bool;
      Especial_M351 : Bool;
      Bit_02_M351 : Bool;
      Retroceder_M351 : Bool;
      Retirar_M351 : Bool;
      Continuar_M351 : Bool;
      Entrar_M351 : Bool;
      EmiOK_M351 : Bool;
      FinLote_M352 : Bool;
      Especial_M352 : Bool;
      Bit_02_M352 : Bool;
      Retroceder_M352 : Bool;
      Retirar_M352 : Bool;
      Continuar_M352 : Bool;
      Entrar_M352 : Bool;
      EmiOK_M352 : Bool;
      FinLote_M353 : Bool;
      Especial_M353 : Bool;
      Bit_02_M353 : Bool;
      Retroceder_M353 : Bool;
      Retirar_M353 : Bool;
      Continuar_M353 : Bool;
      Entrar_M353 : Bool;
      EmiOK_M353 : Bool;
      FinLote_M354 : Bool;
      Especial_M354 : Bool;
      Bit_02_M354 : Bool;
      Retroceder_M354 : Bool;
      Retirar_M354 : Bool;
      Continuar_M354 : Bool;
      Entrar_M354 : Bool;
      EmiOK_M354 : Bool;
      FinLote_M355 : Bool;
      Especial_M355 : Bool;
      Bit_02_M355 : Bool;
      Retroceder_M355 : Bool;
      Retirar_M355 : Bool;
      Continuar_M355 : Bool;
      Entrar_M355 : Bool;
      EmiOK_M355 : Bool;
      FinLote_M356 : Bool;
      Especial_M356 : Bool;
      Bit_02_M356 : Bool;
      Retroceder_M356 : Bool;
      Retirar_M356 : Bool;
      Continuar_M356 : Bool;
      Entrar_M356 : Bool;
      EmiOK_M356 : Bool;
      FinLote_M357 : Bool;
      Especial_M357 : Bool;
      Bit_02_M357 : Bool;
      Retroceder_M357 : Bool;
      Retirar_M357 : Bool;
      Continuar_M357 : Bool;
      Entrar_M357 : Bool;
      EmiOK_M357 : Bool;
      FinLote_M358 : Bool;
      Especial_M358 : Bool;
      Bit_02_M358 : Bool;
      Retroceder_M358 : Bool;
      Retirar_M358 : Bool;
      Continuar_M358 : Bool;
      Entrar_M358 : Bool;
      EmiOK_M358 : Bool;
      FinLote_M359 : Bool;
      Especial_M359 : Bool;
      Bit_02_M359 : Bool;
      Retroceder_M359 : Bool;
      Retirar_M359 : Bool;
      Continuar_M359 : Bool;
      Entrar_M359 : Bool;
      EmiOK_M359 : Bool;
      FinLote_M360 : Bool;
      Especial_M360 : Bool;
      Bit_02_M360 : Bool;
      Retroceder_M360 : Bool;
      Retirar_M360 : Bool;
      Continuar_M360 : Bool;
      Entrar_M360 : Bool;
      EmiOK_M360 : Bool;
      FinLote_M361 : Bool;
      Especial_M361 : Bool;
      Bit_02_M361 : Bool;
      Retroceder_M361 : Bool;
      Retirar_M361 : Bool;
      Continuar_M361 : Bool;
      Entrar_M361 : Bool;
      EmiOK_M361 : Bool;
      FinLote_M362 : Bool;
      Especial_M362 : Bool;
      Bit_02_M362 : Bool;
      Retroceder_M362 : Bool;
      Retirar_M362 : Bool;
      Continuar_M362 : Bool;
      Entrar_M362 : Bool;
      EmiOK_M362 : Bool;
      FinLote_M363 : Bool;
      Especial_M363 : Bool;
      Bit_02_M363 : Bool;
      Retroceder_M363 : Bool;
      Retirar_M363 : Bool;
      Continuar_M363 : Bool;
      Entrar_M363 : Bool;
      EmiOK_M363 : Bool;
      FinLote_M364 : Bool;
      Especial_M364 : Bool;
      Bit_02_M364 : Bool;
      Retroceder_M364 : Bool;
      Retirar_M364 : Bool;
      Continuar_M364 : Bool;
      Entrar_M364 : Bool;
      EmiOK_M364 : Bool;
      FinLote_M365 : Bool;
      Especial_M365 : Bool;
      Bit_02_M365 : Bool;
      Retroceder_M365 : Bool;
      Retirar_M365 : Bool;
      Continuar_M365 : Bool;
      Entrar_M365 : Bool;
      EmiOK_M365 : Bool;
      FinLote_M366 : Bool;
      Especial_M366 : Bool;
      Bit_02_M366 : Bool;
      Retroceder_M366 : Bool;
      Retirar_M366 : Bool;
      Continuar_M366 : Bool;
      Entrar_M366 : Bool;
      EmiOK_M366 : Bool;
      FinLote_M367 : Bool;
      Especial_M367 : Bool;
      Bit_02_M367 : Bool;
      Retroceder_M367 : Bool;
      Retirar_M367 : Bool;
      Continuar_M367 : Bool;
      Entrar_M367 : Bool;
      EmiOK_M367 : Bool;
      FinLote_M368 : Bool;
      Especial_M368 : Bool;
      Bit_02_M368 : Bool;
      Retroceder_M368 : Bool;
      Retirar_M368 : Bool;
      Continuar_M368 : Bool;
      Entrar_M368 : Bool;
      EmiOK_M368 : Bool;
      FinLote_M369 : Bool;
      Especial_M369 : Bool;
      Bit_02_M369 : Bool;
      Retroceder_M369 : Bool;
      Retirar_M369 : Bool;
      Continuar_M369 : Bool;
      Entrar_M369 : Bool;
      EmiOK_M369 : Bool;
      FinLote_M370 : Bool;
      Especial_M370 : Bool;
      Bit_02_M370 : Bool;
      Retroceder_M370 : Bool;
      Retirar_M370 : Bool;
      Continuar_M370 : Bool;
      Entrar_M370 : Bool;
      EmiOK_M370 : Bool;
      FinLote_M371 : Bool;
      Especial_M371 : Bool;
      Bit_02_M371 : Bool;
      Retroceder_M371 : Bool;
      Retirar_M371 : Bool;
      Continuar_M371 : Bool;
      Entrar_M371 : Bool;
      EmiOK_M371 : Bool;
      FinLote_M372 : Bool;
      Especial_M372 : Bool;
      Bit_02_M372 : Bool;
      Retroceder_M372 : Bool;
      Retirar_M372 : Bool;
      Continuar_M372 : Bool;
      Entrar_M372 : Bool;
      EmiOK_M372 : Bool;
      FinLote_M373 : Bool;
      Especial_M373 : Bool;
      Bit_02_M373 : Bool;
      Retroceder_M373 : Bool;
      Retirar_M373 : Bool;
      Continuar_M373 : Bool;
      Entrar_M373 : Bool;
      EmiOK_M373 : Bool;
      FinLote_M374 : Bool;
      Especial_M374 : Bool;
      Bit_02_M374 : Bool;
      Retroceder_M374 : Bool;
      Retirar_M374 : Bool;
      Continuar_M374 : Bool;
      Entrar_M374 : Bool;
      EmiOK_M374 : Bool;
      FinLote_M375 : Bool;
      Especial_M375 : Bool;
      Bit_02_M375 : Bool;
      Retroceder_M375 : Bool;
      Retirar_M375 : Bool;
      Continuar_M375 : Bool;
      Entrar_M375 : Bool;
      EmiOK_M375 : Bool;
      FinLote_M376 : Bool;
      Especial_M376 : Bool;
      Bit_02_M376 : Bool;
      Retroceder_M376 : Bool;
      Retirar_M376 : Bool;
      Continuar_M376 : Bool;
      Entrar_M376 : Bool;
      EmiOK_M376 : Bool;
      FinLote_M377 : Bool;
      Especial_M377 : Bool;
      Bit_02_M377 : Bool;
      Retroceder_M377 : Bool;
      Retirar_M377 : Bool;
      Continuar_M377 : Bool;
      Entrar_M377 : Bool;
      EmiOK_M377 : Bool;
      FinLote_M378 : Bool;
      Especial_M378 : Bool;
      Bit_02_M378 : Bool;
      Retroceder_M378 : Bool;
      Retirar_M378 : Bool;
      Continuar_M378 : Bool;
      Entrar_M378 : Bool;
      EmiOK_M378 : Bool;
      FinLote_M379 : Bool;
      Especial_M379 : Bool;
      Bit_02_M379 : Bool;
      Retroceder_M379 : Bool;
      Retirar_M379 : Bool;
      Continuar_M379 : Bool;
      Entrar_M379 : Bool;
      EmiOK_M379 : Bool;
      FinLote_M380 : Bool;
      Especial_M380 : Bool;
      Bit_02_M380 : Bool;
      Retroceder_M380 : Bool;
      Retirar_M380 : Bool;
      Continuar_M380 : Bool;
      Entrar_M380 : Bool;
      EmiOK_M380 : Bool;
      FinLote_M381 : Bool;
      Especial_M381 : Bool;
      Bit_02_M381 : Bool;
      Retroceder_M381 : Bool;
      Retirar_M381 : Bool;
      Continuar_M381 : Bool;
      Entrar_M381 : Bool;
      EmiOK_M381 : Bool;
      FinLote_M382 : Bool;
      Especial_M382 : Bool;
      Bit_02_M382 : Bool;
      Retroceder_M382 : Bool;
      Retirar_M382 : Bool;
      Continuar_M382 : Bool;
      Entrar_M382 : Bool;
      EmiOK_M382 : Bool;
      FinLote_M383 : Bool;
      Especial_M383 : Bool;
      Bit_02_M383 : Bool;
      Retroceder_M383 : Bool;
      Retirar_M383 : Bool;
      Continuar_M383 : Bool;
      Entrar_M383 : Bool;
      EmiOK_M383 : Bool;
      FinLote_M384 : Bool;
      Especial_M384 : Bool;
      Bit_02_M384 : Bool;
      Retroceder_M384 : Bool;
      Retirar_M384 : Bool;
      Continuar_M384 : Bool;
      Entrar_M384 : Bool;
      EmiOK_M384 : Bool;
      FinLote_M385 : Bool;
      Especial_M385 : Bool;
      Bit_02_M385 : Bool;
      Retroceder_M385 : Bool;
      Retirar_M385 : Bool;
      Continuar_M385 : Bool;
      Entrar_M385 : Bool;
      EmiOK_M385 : Bool;
      FinLote_M386 : Bool;
      Especial_M386 : Bool;
      Bit_02_M386 : Bool;
      Retroceder_M386 : Bool;
      Retirar_M386 : Bool;
      Continuar_M386 : Bool;
      Entrar_M386 : Bool;
      EmiOK_M386 : Bool;
      FinLote_M387 : Bool;
      Especial_M387 : Bool;
      Bit_02_M387 : Bool;
      Retroceder_M387 : Bool;
      Retirar_M387 : Bool;
      Continuar_M387 : Bool;
      Entrar_M387 : Bool;
      EmiOK_M387 : Bool;
      FinLote_M388 : Bool;
      Especial_M388 : Bool;
      Bit_02_M388 : Bool;
      Retroceder_M388 : Bool;
      Retirar_M388 : Bool;
      Continuar_M388 : Bool;
      Entrar_M388 : Bool;
      EmiOK_M388 : Bool;
      FinLote_M389 : Bool;
      Especial_M389 : Bool;
      Bit_02_M389 : Bool;
      Retroceder_M389 : Bool;
      Retirar_M389 : Bool;
      Continuar_M389 : Bool;
      Entrar_M389 : Bool;
      EmiOK_M389 : Bool;
      FinLote_M390 : Bool;
      Especial_M390 : Bool;
      Bit_02_M390 : Bool;
      Retroceder_M390 : Bool;
      Retirar_M390 : Bool;
      Continuar_M390 : Bool;
      Entrar_M390 : Bool;
      EmiOK_M390 : Bool;
      FinLote_M391 : Bool;
      Especial_M391 : Bool;
      Bit_02_M391 : Bool;
      Retroceder_M391 : Bool;
      Retirar_M391 : Bool;
      Continuar_M391 : Bool;
      Entrar_M391 : Bool;
      EmiOK_M391 : Bool;
      FinLote_M392 : Bool;
      Especial_M392 : Bool;
      Bit_02_M392 : Bool;
      Retroceder_M392 : Bool;
      Retirar_M392 : Bool;
      Continuar_M392 : Bool;
      Entrar_M392 : Bool;
      EmiOK_M392 : Bool;
      FinLote_M393 : Bool;
      Especial_M393 : Bool;
      Bit_02_M393 : Bool;
      Retroceder_M393 : Bool;
      Retirar_M393 : Bool;
      Continuar_M393 : Bool;
      Entrar_M393 : Bool;
      EmiOK_M393 : Bool;
      FinLote_M394 : Bool;
      Especial_M394 : Bool;
      Bit_02_M394 : Bool;
      Retroceder_M394 : Bool;
      Retirar_M394 : Bool;
      Continuar_M394 : Bool;
      Entrar_M394 : Bool;
      EmiOK_M394 : Bool;
      FinLote_M395 : Bool;
      Especial_M395 : Bool;
      Bit_02_M395 : Bool;
      Retroceder_M395 : Bool;
      Retirar_M395 : Bool;
      Continuar_M395 : Bool;
      Entrar_M395 : Bool;
      EmiOK_M395 : Bool;
      FinLote_M396 : Bool;
      Especial_M396 : Bool;
      Bit_02_M396 : Bool;
      Retroceder_M396 : Bool;
      Retirar_M396 : Bool;
      Continuar_M396 : Bool;
      Entrar_M396 : Bool;
      EmiOK_M396 : Bool;
      FinLote_M397 : Bool;
      Especial_M397 : Bool;
      Bit_02_M397 : Bool;
      Retroceder_M397 : Bool;
      Retirar_M397 : Bool;
      Continuar_M397 : Bool;
      Entrar_M397 : Bool;
      EmiOK_M397 : Bool;
      FinLote_M398 : Bool;
      Especial_M398 : Bool;
      Bit_02_M398 : Bool;
      Retroceder_M398 : Bool;
      Retirar_M398 : Bool;
      Continuar_M398 : Bool;
      Entrar_M398 : Bool;
      EmiOK_M398 : Bool;
      FinLote_M399 : Bool;
      Especial_M399 : Bool;
      Bit_02_M399 : Bool;
      Retroceder_M399 : Bool;
      Retirar_M399 : Bool;
      Continuar_M399 : Bool;
      Entrar_M399 : Bool;
      EmiOK_M399 : Bool;
      FinLote_M400 : Bool;
      Especial_M400 : Bool;
      Bit_02_M400 : Bool;
      Retroceder_M400 : Bool;
      Retirar_M400 : Bool;
      Continuar_M400 : Bool;
      Entrar_M400 : Bool;
      EmiOK_M400 : Bool;
      FinLote_M401 : Bool;
      Especial_M401 : Bool;
      Bit_02_M401 : Bool;
      Retroceder_M401 : Bool;
      Retirar_M401 : Bool;
      Continuar_M401 : Bool;
      Entrar_M401 : Bool;
      EmiOK_M401 : Bool;
      FinLote_M402 : Bool;
      Especial_M402 : Bool;
      Bit_02_M402 : Bool;
      Retroceder_M402 : Bool;
      Retirar_M402 : Bool;
      Continuar_M402 : Bool;
      Entrar_M402 : Bool;
      EmiOK_M402 : Bool;
      FinLote_M403 : Bool;
      Especial_M403 : Bool;
      Bit_02_M403 : Bool;
      Retroceder_M403 : Bool;
      Retirar_M403 : Bool;
      Continuar_M403 : Bool;
      Entrar_M403 : Bool;
      EmiOK_M403 : Bool;
      FinLote_M404 : Bool;
      Especial_M404 : Bool;
      Bit_02_M404 : Bool;
      Retroceder_M404 : Bool;
      Retirar_M404 : Bool;
      Continuar_M404 : Bool;
      Entrar_M404 : Bool;
      EmiOK_M404 : Bool;
      FinLote_M405 : Bool;
      Especial_M405 : Bool;
      Bit_02_M405 : Bool;
      Retroceder_M405 : Bool;
      Retirar_M405 : Bool;
      Continuar_M405 : Bool;
      Entrar_M405 : Bool;
      EmiOK_M405 : Bool;
      FinLote_M406 : Bool;
      Especial_M406 : Bool;
      Bit_02_M406 : Bool;
      Retroceder_M406 : Bool;
      Retirar_M406 : Bool;
      Continuar_M406 : Bool;
      Entrar_M406 : Bool;
      EmiOK_M406 : Bool;
      FinLote_M407 : Bool;
      Especial_M407 : Bool;
      Bit_02_M407 : Bool;
      Retroceder_M407 : Bool;
      Retirar_M407 : Bool;
      Continuar_M407 : Bool;
      Entrar_M407 : Bool;
      EmiOK_M407 : Bool;
      FinLote_M408 : Bool;
      Especial_M408 : Bool;
      Bit_02_M408 : Bool;
      Retroceder_M408 : Bool;
      Retirar_M408 : Bool;
      Continuar_M408 : Bool;
      Entrar_M408 : Bool;
      EmiOK_M408 : Bool;
      FinLote_M409 : Bool;
      Especial_M409 : Bool;
      Bit_02_M409 : Bool;
      Retroceder_M409 : Bool;
      Retirar_M409 : Bool;
      Continuar_M409 : Bool;
      Entrar_M409 : Bool;
      EmiOK_M409 : Bool;
      FinLote_M410 : Bool;
      Especial_M410 : Bool;
      Bit_02_M410 : Bool;
      Retroceder_M410 : Bool;
      Retirar_M410 : Bool;
      Continuar_M410 : Bool;
      Entrar_M410 : Bool;
      EmiOK_M410 : Bool;
      FinLote_M411 : Bool;
      Especial_M411 : Bool;
      Bit_02_M411 : Bool;
      Retroceder_M411 : Bool;
      Retirar_M411 : Bool;
      Continuar_M411 : Bool;
      Entrar_M411 : Bool;
      EmiOK_M411 : Bool;
      FinLote_M412 : Bool;
      Especial_M412 : Bool;
      Bit_02_M412 : Bool;
      Retroceder_M412 : Bool;
      Retirar_M412 : Bool;
      Continuar_M412 : Bool;
      Entrar_M412 : Bool;
      EmiOK_M412 : Bool;
      FinLote_M413 : Bool;
      Especial_M413 : Bool;
      Bit_02_M413 : Bool;
      Retroceder_M413 : Bool;
      Retirar_M413 : Bool;
      Continuar_M413 : Bool;
      Entrar_M413 : Bool;
      EmiOK_M413 : Bool;
      FinLote_M414 : Bool;
      Especial_M414 : Bool;
      Bit_02_M414 : Bool;
      Retroceder_M414 : Bool;
      Retirar_M414 : Bool;
      Continuar_M414 : Bool;
      Entrar_M414 : Bool;
      EmiOK_M414 : Bool;
      FinLote_M415 : Bool;
      Especial_M415 : Bool;
      Bit_02_M415 : Bool;
      Retroceder_M415 : Bool;
      Retirar_M415 : Bool;
      Continuar_M415 : Bool;
      Entrar_M415 : Bool;
      EmiOK_M415 : Bool;
      FinLote_M416 : Bool;
      Especial_M416 : Bool;
      Bit_02_M416 : Bool;
      Retroceder_M416 : Bool;
      Retirar_M416 : Bool;
      Continuar_M416 : Bool;
      Entrar_M416 : Bool;
      EmiOK_M416 : Bool;
      FinLote_M417 : Bool;
      Especial_M417 : Bool;
      Bit_02_M417 : Bool;
      Retroceder_M417 : Bool;
      Retirar_M417 : Bool;
      Continuar_M417 : Bool;
      Entrar_M417 : Bool;
      EmiOK_M417 : Bool;
      FinLote_M418 : Bool;
      Especial_M418 : Bool;
      Bit_02_M418 : Bool;
      Retroceder_M418 : Bool;
      Retirar_M418 : Bool;
      Continuar_M418 : Bool;
      Entrar_M418 : Bool;
      EmiOK_M418 : Bool;
      FinLote_M419 : Bool;
      Especial_M419 : Bool;
      Bit_02_M419 : Bool;
      Retroceder_M419 : Bool;
      Retirar_M419 : Bool;
      Continuar_M419 : Bool;
      Entrar_M419 : Bool;
      EmiOK_M419 : Bool;
      FinLote_M420 : Bool;
      Especial_M420 : Bool;
      Bit_02_M420 : Bool;
      Retroceder_M420 : Bool;
      Retirar_M420 : Bool;
      Continuar_M420 : Bool;
      Entrar_M420 : Bool;
      EmiOK_M420 : Bool;
      FinLote_M421 : Bool;
      Especial_M421 : Bool;
      Bit_02_M421 : Bool;
      Retroceder_M421 : Bool;
      Retirar_M421 : Bool;
      Continuar_M421 : Bool;
      Entrar_M421 : Bool;
      EmiOK_M421 : Bool;
      FinLote_M422 : Bool;
      Especial_M422 : Bool;
      Bit_02_M422 : Bool;
      Retroceder_M422 : Bool;
      Retirar_M422 : Bool;
      Continuar_M422 : Bool;
      Entrar_M422 : Bool;
      EmiOK_M422 : Bool;
      FinLote_M423 : Bool;
      Especial_M423 : Bool;
      Bit_02_M423 : Bool;
      Retroceder_M423 : Bool;
      Retirar_M423 : Bool;
      Continuar_M423 : Bool;
      Entrar_M423 : Bool;
      EmiOK_M423 : Bool;
      FinLote_M424 : Bool;
      Especial_M424 : Bool;
      Bit_02_M424 : Bool;
      Retroceder_M424 : Bool;
      Retirar_M424 : Bool;
      Continuar_M424 : Bool;
      Entrar_M424 : Bool;
      EmiOK_M424 : Bool;
      FinLote_M425 : Bool;
      Especial_M425 : Bool;
      Bit_02_M425 : Bool;
      Retroceder_M425 : Bool;
      Retirar_M425 : Bool;
      Continuar_M425 : Bool;
      Entrar_M425 : Bool;
      EmiOK_M425 : Bool;
      FinLote_M426 : Bool;
      Especial_M426 : Bool;
      Bit_02_M426 : Bool;
      Retroceder_M426 : Bool;
      Retirar_M426 : Bool;
      Continuar_M426 : Bool;
      Entrar_M426 : Bool;
      EmiOK_M426 : Bool;
      FinLote_M427 : Bool;
      Especial_M427 : Bool;
      Bit_02_M427 : Bool;
      Retroceder_M427 : Bool;
      Retirar_M427 : Bool;
      Continuar_M427 : Bool;
      Entrar_M427 : Bool;
      EmiOK_M427 : Bool;
      FinLote_M428 : Bool;
      Especial_M428 : Bool;
      Bit_02_M428 : Bool;
      Retroceder_M428 : Bool;
      Retirar_M428 : Bool;
      Continuar_M428 : Bool;
      Entrar_M428 : Bool;
      EmiOK_M428 : Bool;
      FinLote_M429 : Bool;
      Especial_M429 : Bool;
      Bit_02_M429 : Bool;
      Retroceder_M429 : Bool;
      Retirar_M429 : Bool;
      Continuar_M429 : Bool;
      Entrar_M429 : Bool;
      EmiOK_M429 : Bool;
      FinLote_M430 : Bool;
      Especial_M430 : Bool;
      Bit_02_M430 : Bool;
      Retroceder_M430 : Bool;
      Retirar_M430 : Bool;
      Continuar_M430 : Bool;
      Entrar_M430 : Bool;
      EmiOK_M430 : Bool;
      FinLote_M431 : Bool;
      Especial_M431 : Bool;
      Bit_02_M431 : Bool;
      Retroceder_M431 : Bool;
      Retirar_M431 : Bool;
      Continuar_M431 : Bool;
      Entrar_M431 : Bool;
      EmiOK_M431 : Bool;
      FinLote_M432 : Bool;
      Especial_M432 : Bool;
      Bit_02_M432 : Bool;
      Retroceder_M432 : Bool;
      Retirar_M432 : Bool;
      Continuar_M432 : Bool;
      Entrar_M432 : Bool;
      EmiOK_M432 : Bool;
      FinLote_M433 : Bool;
      Especial_M433 : Bool;
      Bit_02_M433 : Bool;
      Retroceder_M433 : Bool;
      Retirar_M433 : Bool;
      Continuar_M433 : Bool;
      Entrar_M433 : Bool;
      EmiOK_M433 : Bool;
      FinLote_M434 : Bool;
      Especial_M434 : Bool;
      Bit_02_M434 : Bool;
      Retroceder_M434 : Bool;
      Retirar_M434 : Bool;
      Continuar_M434 : Bool;
      Entrar_M434 : Bool;
      EmiOK_M434 : Bool;
      FinLote_M435 : Bool;
      Especial_M435 : Bool;
      Bit_02_M435 : Bool;
      Retroceder_M435 : Bool;
      Retirar_M435 : Bool;
      Continuar_M435 : Bool;
      Entrar_M435 : Bool;
      EmiOK_M435 : Bool;
      FinLote_M436 : Bool;
      Especial_M436 : Bool;
      Bit_02_M436 : Bool;
      Retroceder_M436 : Bool;
      Retirar_M436 : Bool;
      Continuar_M436 : Bool;
      Entrar_M436 : Bool;
      EmiOK_M436 : Bool;
      FinLote_M437 : Bool;
      Especial_M437 : Bool;
      Bit_02_M437 : Bool;
      Retroceder_M437 : Bool;
      Retirar_M437 : Bool;
      Continuar_M437 : Bool;
      Entrar_M437 : Bool;
      EmiOK_M437 : Bool;
      FinLote_M438 : Bool;
      Especial_M438 : Bool;
      Bit_02_M438 : Bool;
      Retroceder_M438 : Bool;
      Retirar_M438 : Bool;
      Continuar_M438 : Bool;
      Entrar_M438 : Bool;
      EmiOK_M438 : Bool;
      FinLote_M439 : Bool;
      Especial_M439 : Bool;
      Bit_02_M439 : Bool;
      Retroceder_M439 : Bool;
      Retirar_M439 : Bool;
      Continuar_M439 : Bool;
      Entrar_M439 : Bool;
      EmiOK_M439 : Bool;
      FinLote_M440 : Bool;
      Especial_M440 : Bool;
      Bit_02_M440 : Bool;
      Retroceder_M440 : Bool;
      Retirar_M440 : Bool;
      Continuar_M440 : Bool;
      Entrar_M440 : Bool;
      EmiOK_M440 : Bool;
      FinLote_M441 : Bool;
      Especial_M441 : Bool;
      Bit_02_M441 : Bool;
      Retroceder_M441 : Bool;
      Retirar_M441 : Bool;
      Continuar_M441 : Bool;
      Entrar_M441 : Bool;
      EmiOK_M441 : Bool;
      FinLote_M442 : Bool;
      Especial_M442 : Bool;
      Bit_02_M442 : Bool;
      Retroceder_M442 : Bool;
      Retirar_M442 : Bool;
      Continuar_M442 : Bool;
      Entrar_M442 : Bool;
      EmiOK_M442 : Bool;
      FinLote_M443 : Bool;
      Especial_M443 : Bool;
      Bit_02_M443 : Bool;
      Retroceder_M443 : Bool;
      Retirar_M443 : Bool;
      Continuar_M443 : Bool;
      Entrar_M443 : Bool;
      EmiOK_M443 : Bool;
      FinLote_M444 : Bool;
      Especial_M444 : Bool;
      Bit_02_M444 : Bool;
      Retroceder_M444 : Bool;
      Retirar_M444 : Bool;
      Continuar_M444 : Bool;
      Entrar_M444 : Bool;
      EmiOK_M444 : Bool;
      FinLote_M445 : Bool;
      Especial_M445 : Bool;
      Bit_02_M445 : Bool;
      Retroceder_M445 : Bool;
      Retirar_M445 : Bool;
      Continuar_M445 : Bool;
      Entrar_M445 : Bool;
      EmiOK_M445 : Bool;
      FinLote_M446 : Bool;
      Especial_M446 : Bool;
      Bit_02_M446 : Bool;
      Retroceder_M446 : Bool;
      Retirar_M446 : Bool;
      Continuar_M446 : Bool;
      Entrar_M446 : Bool;
      EmiOK_M446 : Bool;
      FinLote_M447 : Bool;
      Especial_M447 : Bool;
      Bit_02_M447 : Bool;
      Retroceder_M447 : Bool;
      Retirar_M447 : Bool;
      Continuar_M447 : Bool;
      Entrar_M447 : Bool;
      EmiOK_M447 : Bool;
      FinLote_M448 : Bool;
      Especial_M448 : Bool;
      Bit_02_M448 : Bool;
      Retroceder_M448 : Bool;
      Retirar_M448 : Bool;
      Continuar_M448 : Bool;
      Entrar_M448 : Bool;
      EmiOK_M448 : Bool;
      FinLote_M449 : Bool;
      Especial_M449 : Bool;
      Bit_02_M449 : Bool;
      Retroceder_M449 : Bool;
      Retirar_M449 : Bool;
      Continuar_M449 : Bool;
      Entrar_M449 : Bool;
      EmiOK_M449 : Bool;
      FinLote_M450 : Bool;
      Especial_M450 : Bool;
      Bit_02_M450 : Bool;
      Retroceder_M450 : Bool;
      Retirar_M450 : Bool;
      Continuar_M450 : Bool;
      Entrar_M450 : Bool;
      EmiOK_M450 : Bool;
      FinLote_M451 : Bool;
      Especial_M451 : Bool;
      Bit_02_M451 : Bool;
      Retroceder_M451 : Bool;
      Retirar_M451 : Bool;
      Continuar_M451 : Bool;
      Entrar_M451 : Bool;
      EmiOK_M451 : Bool;
      FinLote_M452 : Bool;
      Especial_M452 : Bool;
      Bit_02_M452 : Bool;
      Retroceder_M452 : Bool;
      Retirar_M452 : Bool;
      Continuar_M452 : Bool;
      Entrar_M452 : Bool;
      EmiOK_M452 : Bool;
      FinLote_M453 : Bool;
      Especial_M453 : Bool;
      Bit_02_M453 : Bool;
      Retroceder_M453 : Bool;
      Retirar_M453 : Bool;
      Continuar_M453 : Bool;
      Entrar_M453 : Bool;
      EmiOK_M453 : Bool;
      FinLote_M454 : Bool;
      Especial_M454 : Bool;
      Bit_02_M454 : Bool;
      Retroceder_M454 : Bool;
      Retirar_M454 : Bool;
      Continuar_M454 : Bool;
      Entrar_M454 : Bool;
      EmiOK_M454 : Bool;
      FinLote_M455 : Bool;
      Especial_M455 : Bool;
      Bit_02_M455 : Bool;
      Retroceder_M455 : Bool;
      Retirar_M455 : Bool;
      Continuar_M455 : Bool;
      Entrar_M455 : Bool;
      EmiOK_M455 : Bool;
      FinLote_M456 : Bool;
      Especial_M456 : Bool;
      Bit_02_M456 : Bool;
      Retroceder_M456 : Bool;
      Retirar_M456 : Bool;
      Continuar_M456 : Bool;
      Entrar_M456 : Bool;
      EmiOK_M456 : Bool;
      FinLote_M457 : Bool;
      Especial_M457 : Bool;
      Bit_02_M457 : Bool;
      Retroceder_M457 : Bool;
      Retirar_M457 : Bool;
      Continuar_M457 : Bool;
      Entrar_M457 : Bool;
      EmiOK_M457 : Bool;
      FinLote_M458 : Bool;
      Especial_M458 : Bool;
      Bit_02_M458 : Bool;
      Retroceder_M458 : Bool;
      Retirar_M458 : Bool;
      Continuar_M458 : Bool;
      Entrar_M458 : Bool;
      EmiOK_M458 : Bool;
      FinLote_M459 : Bool;
      Especial_M459 : Bool;
      Bit_02_M459 : Bool;
      Retroceder_M459 : Bool;
      Retirar_M459 : Bool;
      Continuar_M459 : Bool;
      Entrar_M459 : Bool;
      EmiOK_M459 : Bool;
      FinLote_M460 : Bool;
